// TwinCAT 3 PLC project plc_kfe_gatt
// ProgramVersion: 3.1.4023.0
// libraries:
//   LCLS General, * (SLAC)
//   lcls-twincat-motion, * (SLAC)
//   lcls-twincat-vacuum, * (SLAC)
//   PMPS, * (SLAC - LCLS)
//   Tc2_ControllerToolbox, * (Beckhoff Automation GmbH)
//   Tc2_EtherCAT, * (Beckhoff Automation GmbH)
//   Tc2_MC2, * (Beckhoff Automation GmbH)
//   Tc2_Standard, * (Beckhoff Automation GmbH)
//   Tc2_System, * (Beckhoff Automation GmbH)
//   Tc2_Utilities, * (Beckhoff Automation GmbH)
//   Tc3_JsonXml, * (Beckhoff Automation GmbH)
//   Tc3_Module, * (Beckhoff Automation GmbH)
//   TcUnit, * (www.tcunit.org)
// project tree:
//   DUTs/ E_HomeState.TcDUT (not stored), E_MAA_States.TcDUT (not stored), E_MoveState.TcDUT (not stored), ST_VGP.TcDUT (not stored)
//   GVLs/ GVL_Devices.TcGVL, GVL_GATT.TcGVL (not stored), GVL_ILK.TcGVL, GVL_MOT.TcGVL (not stored), GVL_Variables.TcGVL (not stored), Main.TcGVL (not stored)
//   / PlcTask.TcTTO (not stored)
//   POUs/ DIAGNOSTICS.TcPOU, FB_MAA.TcPOU, FB_MAA_States.TcPOU, FB_VGP.TcPOU, PRG_1_PlcTask.TcPOU, PRG_GATT.TcPOU, PRG_ILK.TcPOU, PRG_INJ.TcPOU, PRG_Motion.TcPOU, PRG_Motors_Test.TcPOU (not stored), PRG_VGP.TcPOU (not stored)
//   POUs/Test/ FB_ILK_TEST.TcPOU
// real-time tasks:
//   TASK PlcTask: cycle T#10ms, priority 20, ADS port 350
// motion (NC):
//   TASK NC-Task 1 SAF: cycle T#2ms, priority 4, ADS port 501
//   TASK NC-Task 1 SVB: cycle T#10ms, priority 8, ADS port 511
//   AXIS MA_1_X (id 1)
//     Velo: Maximum=5
//     OtherSettings: AllowMotionCmdToSlave=true
//     encoder EncType=4
//       EncPara: ScaleFactorNumerator=6.1991875e-05, MaxCount=#x0000ffff
//         Inc: RefSoftSyncMask=#x0000ffff
//     drive DrvType=24
//       Analog: VeloReferenz=7.93496, TorqueScale=10, ScaleFactorActTorque=0.1
//       TimeComp: TaskDelayCycles=1
//     controller CtrType=1
//       CtrPara: PriorControlFactor=1
//         Observer: BandWidth=20
//   AXIS MA_1_Y (id 2)
//     Dynamic: AccelerationMaximum=30, DecelerationMaximum=30
//     Velo: Maximum=40
//     OtherSettings: AllowMotionCmdToSlave=true
//     encoder EncType=7
//       EncPara: ScaleFactorNumerator=0.001452636719, Offset=-47.5985, MaxCount=#x0000ffff, ReferenceSystem=1
//         Inc: RefSoftSyncMask=#x0000ffff
//     drive DrvType=24
//       Analog: VeloReferenz=50, TorqueScale=10, ScaleFactorActTorque=0.1
//       TimeComp: TaskDelayCycles=1
//     controller CtrType=1
//       CtrPara: PriorControlFactor=1
//         Observer: BandWidth=20
//   AXIS MA_2_X (id 3)
//     Velo: Maximum=5
//     OtherSettings: AllowMotionCmdToSlave=true
//     encoder EncType=4
//       EncPara: ScaleFactorNumerator=6.1991875e-05, MaxCount=#x0000ffff
//         Inc: RefSoftSyncMask=#x0000ffff
//     drive DrvType=24
//       Analog: VeloReferenz=7.93496, TorqueScale=10, ScaleFactorActTorque=0.1
//       TimeComp: TaskDelayCycles=1
//     controller CtrType=1
//       CtrPara: PriorControlFactor=1
//         Observer: BandWidth=20
//   AXIS MA_2_Y (id 4)
//     Dynamic: AccelerationMaximum=30, DecelerationMaximum=30
//     Velo: Maximum=40
//     OtherSettings: AllowMotionCmdToSlave=true
//     encoder EncType=7
//       EncPara: ScaleFactorNumerator=0.001440429688, Offset=-47.056, MaxCount=#x0000ffff, ReferenceSystem=1
//         Inc: RefSoftSyncMask=#x0000ffff
//     drive DrvType=24
//       Analog: VeloReferenz=50, TorqueScale=10, ScaleFactorActTorque=0.1
//       TimeComp: TaskDelayCycles=1
//     controller CtrType=1
//       CtrPara: PriorControlFactor=1
//         Observer: BandWidth=20
//   AXIS MA_3_X (id 5)
//     Velo: Maximum=5
//     OtherSettings: AllowMotionCmdToSlave=true
//     encoder EncType=4
//       EncPara: ScaleFactorNumerator=6.1991875e-05, MaxCount=#x0000ffff
//         Inc: RefSoftSyncMask=#x0000ffff
//     drive DrvType=24
//       Analog: VeloReferenz=7.93496, TorqueScale=10, ScaleFactorActTorque=0.1
//       TimeComp: TaskDelayCycles=1
//     controller CtrType=1
//       CtrPara: PriorControlFactor=1
//         Observer: BandWidth=20
//   AXIS MA_3_Y (id 6)
//     Dynamic: AccelerationMaximum=30, DecelerationMaximum=30
//     Velo: Maximum=40
//     OtherSettings: AllowMotionCmdToSlave=true
//     encoder EncType=7
//       EncPara: ScaleFactorNumerator=0.001439703369, Offset=-47.15, MaxCount=#x0000ffff, ReferenceSystem=1
//         SoftEndMaxControl: Range=47.2
//         Inc: RefSoftSyncMask=#x0000ffff
//     drive DrvType=24
//       Analog: VeloReferenz=50, TorqueScale=10, ScaleFactorActTorque=0.1
//       TimeComp: TaskDelayCycles=1
//     controller CtrType=1
//       CtrPara: PriorControlFactor=1
//         PosDiffControl: Range=1.5
//         Observer: BandWidth=20
//   AXIS MA_4_X (id 7)
//     Velo: Maximum=5
//     OtherSettings: AllowMotionCmdToSlave=true
//     encoder EncType=4
//       EncPara: ScaleFactorNumerator=6.1991875e-05, MaxCount=#x0000ffff
//         Inc: RefSoftSyncMask=#x0000ffff
//     drive DrvType=24
//       Analog: VeloReferenz=7.93496, TorqueScale=10, ScaleFactorActTorque=0.1
//       TimeComp: TaskDelayCycles=1
//     controller CtrType=1
//       CtrPara: PriorControlFactor=1
//         Observer: BandWidth=20
//   AXIS MA_4_Y (id 8)
//     Dynamic: AccelerationMaximum=30, DecelerationMaximum=30
//     Velo: Maximum=40
//     OtherSettings: AllowMotionCmdToSlave=true
//     encoder EncType=4
//       EncPara: ScaleFactorNumerator=0.000390625, MaxCount=#x0000ffff
//         Inc: RefSoftSyncMask=#x0000ffff
//     drive DrvType=24
//       Analog: VeloReferenz=50, TorqueScale=10, ScaleFactorActTorque=0.1
//       TimeComp: TaskDelayCycles=1
//     controller CtrType=1
//       CtrPara: PriorControlFactor=1
//         Observer: BandWidth=20
//   AXIS VGP_80 (id 9)
//     Velo: Maximum=1800
//     OtherSettings: AllowMotionCmdToSlave=true
//     encoder EncType=4
//       EncPara: ScaleFactorNumerator=0.0390625, Inverse=true, MaxCount=#x0000ffff
//         SoftEndMinControl: Enable=true, Range=-15
//         SoftEndMaxControl: Enable=true, Range=1695
//         Inc: RefSoftSyncMask=#x0000ffff
//     drive DrvType=24
//       Analog: VeloReferenz=2000, TorqueScale=10, ScaleFactorActTorque=0.1
//       TimeComp: TaskDelayCycles=1
//     controller CtrType=1
//       CtrPara: PriorControlFactor=1
//         PosDiffControl: Range=75
//         Observer: BandWidth=20
// I/O:
//   DEVICE =+-CX2020%_2FEtherCAT1
// variable links:
//   NC-Task 1 SAF/Axes/MA_1_X <-> =+-CX2020/EtherCAT1/=+-EK1100_02_00/=+-ES7041_02_05
//     Drive/Inputs/In/nState1 @bit 3 <-> STM Status/Status/Error
//     Drive/Inputs/In/nState1 @bit 5 <-> STM Status/Status/Moving negative
//     Drive/Inputs/In/nState1 @bit 4 <-> STM Status/Status/Moving positive
//     Drive/Inputs/In/nState1 @bit 1 <-> STM Status/Status/Ready
//     Drive/Inputs/In/nState1 <-> STM Status/Status/Ready to enable
//     Drive/Inputs/In/nState1 @bit 6 <-> STM Status/Status/Torque reduced
//     Drive/Inputs/In/nState1 @bit 2 <-> STM Status/Status/Warning
//     Drive/Inputs/In/nState2 @bit 3 <-> STM Status/Status/Digital input 1
//     Drive/Inputs/In/nState2 @bit 4 <-> STM Status/Status/Digital input 2
//     Drive/Inputs/In/nState2 @bit 5 <-> STM Status/Status/Sync error
//     Drive/Inputs/In/nState2 @bit 7 <-> STM Status/Status/TxPDO Toggle
//     Drive/Inputs/In/nState4 @bit 1 <-> WcState/InputToggle
//     Drive/Inputs/In/nState4 <-> WcState/WcState
//     Drive/Outputs/Out/nCtrl1 <-> STM Control/Control/Enable
//     Drive/Outputs/Out/nCtrl1 @bit 2 <-> STM Control/Control/Reduce torque
//     Drive/Outputs/Out/nCtrl1 @bit 1 <-> STM Control/Control/Reset
//     Drive/Outputs/Out/nDataOut2[0] <-> STM Velocity/Velocity
//     Enc/Inputs/In/nDataIn1[0] <-> ENC Status compact/Counter value
//     Enc/Inputs/In/nDataIn2[0] <-> ENC Status compact/Latch value
//     Enc/Inputs/In/nState1 @bit 4 <-> ENC Status compact/Status/Counter overflow
//     Enc/Inputs/In/nState1 @bit 3 <-> ENC Status compact/Status/Counter underflow
//     Enc/Inputs/In/nState1 @bit 7 <-> ENC Status compact/Status/Extrapolation stall
//     Enc/Inputs/In/nState1 <-> ENC Status compact/Status/Latch C valid
//     Enc/Inputs/In/nState1 @bit 1 <-> ENC Status compact/Status/Latch extern valid
//     Enc/Inputs/In/nState1 @bit 2 <-> ENC Status compact/Status/Set counter done
//     Enc/Inputs/In/nState2 @bit 4 <-> ENC Status compact/Status/Status of extern latch
//     Enc/Inputs/In/nState2 <-> ENC Status compact/Status/Status of input A
//     Enc/Inputs/In/nState2 @bit 1 <-> ENC Status compact/Status/Status of input B
//     Enc/Inputs/In/nState2 @bit 2 <-> ENC Status compact/Status/Status of input C
//     Enc/Inputs/In/nState2 @bit 5 <-> ENC Status compact/Status/Sync error
//     Enc/Inputs/In/nState2 @bit 7 <-> ENC Status compact/Status/TxPDO Toggle
//     Enc/Inputs/In/nState4 @bit 1 <-> WcState/InputToggle
//     Enc/Inputs/In/nState4 <-> WcState/WcState
//     Enc/Outputs/Out/nCtrl1 <-> ENC Control compact/Control/Enable latch C
//     Enc/Outputs/Out/nCtrl1 @bit 3 <-> ENC Control compact/Control/Enable latch extern on negative edge
//     Enc/Outputs/Out/nCtrl1 @bit 1 <-> ENC Control compact/Control/Enable latch extern on positive edge
//     Enc/Outputs/Out/nCtrl1 @bit 2 <-> ENC Control compact/Control/Set counter
//     Enc/Outputs/Out/nDataOut1[0] <-> ENC Control compact/Set counter value
//   NC-Task 1 SAF/Axes/MA_1_Y <-> =+-CX2020/EtherCAT1/=+-EK1100_02_00/=+-ES3054_02_17
//     Enc/Inputs/In/nDataIn1[0] <-> AI Standard Channel 2/Value
//     Enc/Inputs/In/nState4 @bit 1 <-> WcState/InputToggle
//     Enc/Inputs/In/nState4 <-> WcState/WcState
//   NC-Task 1 SAF/Axes/MA_1_Y <-> =+-CX2020/EtherCAT1/=+-EK1100_02_00/=+-ES7041_02_06
//     Drive/Inputs/In/nState1 @bit 3 <-> STM Status/Status/Error
//     Drive/Inputs/In/nState1 @bit 5 <-> STM Status/Status/Moving negative
//     Drive/Inputs/In/nState1 @bit 4 <-> STM Status/Status/Moving positive
//     Drive/Inputs/In/nState1 @bit 1 <-> STM Status/Status/Ready
//     Drive/Inputs/In/nState1 <-> STM Status/Status/Ready to enable
//     Drive/Inputs/In/nState1 @bit 6 <-> STM Status/Status/Torque reduced
//     Drive/Inputs/In/nState1 @bit 2 <-> STM Status/Status/Warning
//     Drive/Inputs/In/nState2 @bit 3 <-> STM Status/Status/Digital input 1
//     Drive/Inputs/In/nState2 @bit 4 <-> STM Status/Status/Digital input 2
//     Drive/Inputs/In/nState2 @bit 5 <-> STM Status/Status/Sync error
//     Drive/Inputs/In/nState2 @bit 7 <-> STM Status/Status/TxPDO Toggle
//     Drive/Inputs/In/nState4 @bit 1 <-> WcState/InputToggle
//     Drive/Inputs/In/nState4 <-> WcState/WcState
//     Drive/Outputs/Out/nCtrl1 <-> STM Control/Control/Enable
//     Drive/Outputs/Out/nCtrl1 @bit 2 <-> STM Control/Control/Reduce torque
//     Drive/Outputs/Out/nCtrl1 @bit 1 <-> STM Control/Control/Reset
//     Drive/Outputs/Out/nDataOut2[0] <-> STM Velocity/Velocity
//   NC-Task 1 SAF/Axes/MA_2_X <-> =+-CX2020/EtherCAT1/=+-EK1100_02_00/=+-ES7041_02_09
//     Drive/Inputs/In/nState1 @bit 3 <-> STM Status/Status/Error
//     Drive/Inputs/In/nState1 @bit 5 <-> STM Status/Status/Moving negative
//     Drive/Inputs/In/nState1 @bit 4 <-> STM Status/Status/Moving positive
//     Drive/Inputs/In/nState1 @bit 1 <-> STM Status/Status/Ready
//     Drive/Inputs/In/nState1 <-> STM Status/Status/Ready to enable
//     Drive/Inputs/In/nState1 @bit 6 <-> STM Status/Status/Torque reduced
//     Drive/Inputs/In/nState1 @bit 2 <-> STM Status/Status/Warning
//     Drive/Inputs/In/nState2 @bit 3 <-> STM Status/Status/Digital input 1
//     Drive/Inputs/In/nState2 @bit 4 <-> STM Status/Status/Digital input 2
//     Drive/Inputs/In/nState2 @bit 5 <-> STM Status/Status/Sync error
//     Drive/Inputs/In/nState2 @bit 7 <-> STM Status/Status/TxPDO Toggle
//     Drive/Inputs/In/nState4 @bit 1 <-> WcState/InputToggle
//     Drive/Inputs/In/nState4 <-> WcState/WcState
//     Drive/Outputs/Out/nCtrl1 <-> STM Control/Control/Enable
//     Drive/Outputs/Out/nCtrl1 @bit 2 <-> STM Control/Control/Reduce torque
//     Drive/Outputs/Out/nCtrl1 @bit 1 <-> STM Control/Control/Reset
//     Drive/Outputs/Out/nDataOut2[0] <-> STM Velocity/Velocity
//     Enc/Inputs/In/nDataIn1[0] <-> ENC Status compact/Counter value
//     Enc/Inputs/In/nDataIn2[0] <-> ENC Status compact/Latch value
//     Enc/Inputs/In/nState1 @bit 4 <-> ENC Status compact/Status/Counter overflow
//     Enc/Inputs/In/nState1 @bit 3 <-> ENC Status compact/Status/Counter underflow
//     Enc/Inputs/In/nState1 @bit 7 <-> ENC Status compact/Status/Extrapolation stall
//     Enc/Inputs/In/nState1 <-> ENC Status compact/Status/Latch C valid
//     Enc/Inputs/In/nState1 @bit 1 <-> ENC Status compact/Status/Latch extern valid
//     Enc/Inputs/In/nState1 @bit 2 <-> ENC Status compact/Status/Set counter done
//     Enc/Inputs/In/nState2 @bit 4 <-> ENC Status compact/Status/Status of extern latch
//     Enc/Inputs/In/nState2 <-> ENC Status compact/Status/Status of input A
//     Enc/Inputs/In/nState2 @bit 1 <-> ENC Status compact/Status/Status of input B
//     Enc/Inputs/In/nState2 @bit 2 <-> ENC Status compact/Status/Status of input C
//     Enc/Inputs/In/nState2 @bit 5 <-> ENC Status compact/Status/Sync error
//     Enc/Inputs/In/nState2 @bit 7 <-> ENC Status compact/Status/TxPDO Toggle
//     Enc/Inputs/In/nState4 @bit 1 <-> WcState/InputToggle
//     Enc/Inputs/In/nState4 <-> WcState/WcState
//     Enc/Outputs/Out/nCtrl1 <-> ENC Control compact/Control/Enable latch C
//     Enc/Outputs/Out/nCtrl1 @bit 3 <-> ENC Control compact/Control/Enable latch extern on negative edge
//     Enc/Outputs/Out/nCtrl1 @bit 1 <-> ENC Control compact/Control/Enable latch extern on positive edge
//     Enc/Outputs/Out/nCtrl1 @bit 2 <-> ENC Control compact/Control/Set counter
//     Enc/Outputs/Out/nDataOut1[0] <-> ENC Control compact/Set counter value
//   NC-Task 1 SAF/Axes/MA_2_Y <-> =+-CX2020/EtherCAT1/=+-EK1100_02_00/=+-ES3054_02_17
//     Enc/Inputs/In/nDataIn1[0] <-> AI Standard Channel 4/Value
//     Enc/Inputs/In/nState4 @bit 1 <-> WcState/InputToggle
//     Enc/Inputs/In/nState4 <-> WcState/WcState
//   NC-Task 1 SAF/Axes/MA_2_Y <-> =+-CX2020/EtherCAT1/=+-EK1100_02_00/=+-ES7041_02_10
//     Drive/Inputs/In/nState1 @bit 3 <-> STM Status/Status/Error
//     Drive/Inputs/In/nState1 @bit 5 <-> STM Status/Status/Moving negative
//     Drive/Inputs/In/nState1 @bit 4 <-> STM Status/Status/Moving positive
//     Drive/Inputs/In/nState1 @bit 1 <-> STM Status/Status/Ready
//     Drive/Inputs/In/nState1 <-> STM Status/Status/Ready to enable
//     Drive/Inputs/In/nState1 @bit 6 <-> STM Status/Status/Torque reduced
//     Drive/Inputs/In/nState1 @bit 2 <-> STM Status/Status/Warning
//     Drive/Inputs/In/nState2 @bit 3 <-> STM Status/Status/Digital input 1
//     Drive/Inputs/In/nState2 @bit 4 <-> STM Status/Status/Digital input 2
//     Drive/Inputs/In/nState2 @bit 5 <-> STM Status/Status/Sync error
//     Drive/Inputs/In/nState2 @bit 7 <-> STM Status/Status/TxPDO Toggle
//     Drive/Inputs/In/nState4 @bit 1 <-> WcState/InputToggle
//     Drive/Inputs/In/nState4 <-> WcState/WcState
//     Drive/Outputs/Out/nCtrl1 <-> STM Control/Control/Enable
//     Drive/Outputs/Out/nCtrl1 @bit 2 <-> STM Control/Control/Reduce torque
//     Drive/Outputs/Out/nCtrl1 @bit 1 <-> STM Control/Control/Reset
//     Drive/Outputs/Out/nDataOut2[0] <-> STM Velocity/Velocity
//   NC-Task 1 SAF/Axes/MA_3_X <-> =+-CX2020/EtherCAT1/=+-EK1100_04_00/=+-EL7041_04_07
//     Drive/Inputs/In/nState1 @bit 3 <-> STM Status/Status/Error
//     Drive/Inputs/In/nState1 @bit 5 <-> STM Status/Status/Moving negative
//     Drive/Inputs/In/nState1 @bit 4 <-> STM Status/Status/Moving positive
//     Drive/Inputs/In/nState1 @bit 1 <-> STM Status/Status/Ready
//     Drive/Inputs/In/nState1 <-> STM Status/Status/Ready to enable
//     Drive/Inputs/In/nState1 @bit 6 <-> STM Status/Status/Torque reduced
//     Drive/Inputs/In/nState1 @bit 2 <-> STM Status/Status/Warning
//     Drive/Inputs/In/nState2 @bit 3 <-> STM Status/Status/Digital input 1
//     Drive/Inputs/In/nState2 @bit 4 <-> STM Status/Status/Digital input 2
//     Drive/Inputs/In/nState2 @bit 5 <-> STM Status/Status/Sync error
//     Drive/Inputs/In/nState2 @bit 7 <-> STM Status/Status/TxPDO Toggle
//     Drive/Inputs/In/nState4 @bit 1 <-> WcState/InputToggle
//     Drive/Inputs/In/nState4 <-> WcState/WcState
//     Drive/Outputs/Out/nCtrl1 <-> STM Control/Control/Enable
//     Drive/Outputs/Out/nCtrl1 @bit 2 <-> STM Control/Control/Reduce torque
//     Drive/Outputs/Out/nCtrl1 @bit 1 <-> STM Control/Control/Reset
//     Drive/Outputs/Out/nDataOut2[0] <-> STM Velocity/Velocity
//     Enc/Inputs/In/nDataIn1[0] <-> ENC Status compact/Counter value
//     Enc/Inputs/In/nDataIn2[0] <-> ENC Status compact/Latch value
//     Enc/Inputs/In/nState1 @bit 4 <-> ENC Status compact/Status/Counter overflow
//     Enc/Inputs/In/nState1 @bit 3 <-> ENC Status compact/Status/Counter underflow
//     Enc/Inputs/In/nState1 @bit 7 <-> ENC Status compact/Status/Extrapolation stall
//     Enc/Inputs/In/nState1 <-> ENC Status compact/Status/Latch C valid
//     Enc/Inputs/In/nState1 @bit 1 <-> ENC Status compact/Status/Latch extern valid
//     Enc/Inputs/In/nState1 @bit 2 <-> ENC Status compact/Status/Set counter done
//     Enc/Inputs/In/nState2 @bit 4 <-> ENC Status compact/Status/Status of extern latch
//     Enc/Inputs/In/nState2 <-> ENC Status compact/Status/Status of input A
//     Enc/Inputs/In/nState2 @bit 1 <-> ENC Status compact/Status/Status of input B
//     Enc/Inputs/In/nState2 @bit 2 <-> ENC Status compact/Status/Status of input C
//     Enc/Inputs/In/nState2 @bit 5 <-> ENC Status compact/Status/Sync error
//     Enc/Inputs/In/nState2 @bit 7 <-> ENC Status compact/Status/TxPDO Toggle
//     Enc/Inputs/In/nState4 @bit 1 <-> WcState/InputToggle
//     Enc/Inputs/In/nState4 <-> WcState/WcState
//     Enc/Outputs/Out/nCtrl1 <-> ENC Control compact/Control/Enable latch C
//     Enc/Outputs/Out/nCtrl1 @bit 3 <-> ENC Control compact/Control/Enable latch extern on negative edge
//     Enc/Outputs/Out/nCtrl1 @bit 1 <-> ENC Control compact/Control/Enable latch extern on positive edge
//     Enc/Outputs/Out/nCtrl1 @bit 2 <-> ENC Control compact/Control/Set counter
//     Enc/Outputs/Out/nDataOut1[0] <-> ENC Control compact/Set counter value
//   NC-Task 1 SAF/Axes/MA_3_Y <-> =+-CX2020/EtherCAT1/=+-EK1100_04_00/=+-EL7041_04_08
//     Drive/Inputs/In/nState1 @bit 3 <-> STM Status/Status/Error
//     Drive/Inputs/In/nState1 @bit 5 <-> STM Status/Status/Moving negative
//     Drive/Inputs/In/nState1 @bit 4 <-> STM Status/Status/Moving positive
//     Drive/Inputs/In/nState1 @bit 1 <-> STM Status/Status/Ready
//     Drive/Inputs/In/nState1 <-> STM Status/Status/Ready to enable
//     Drive/Inputs/In/nState1 @bit 6 <-> STM Status/Status/Torque reduced
//     Drive/Inputs/In/nState1 @bit 2 <-> STM Status/Status/Warning
//     Drive/Inputs/In/nState2 @bit 3 <-> STM Status/Status/Digital input 1
//     Drive/Inputs/In/nState2 @bit 4 <-> STM Status/Status/Digital input 2
//     Drive/Inputs/In/nState2 @bit 5 <-> STM Status/Status/Sync error
//     Drive/Inputs/In/nState2 @bit 7 <-> STM Status/Status/TxPDO Toggle
//     Drive/Inputs/In/nState4 @bit 1 <-> WcState/InputToggle
//     Drive/Inputs/In/nState4 <-> WcState/WcState
//     Drive/Outputs/Out/nCtrl1 <-> STM Control/Control/Enable
//     Drive/Outputs/Out/nCtrl1 @bit 2 <-> STM Control/Control/Reduce torque
//     Drive/Outputs/Out/nCtrl1 @bit 1 <-> STM Control/Control/Reset
//     Drive/Outputs/Out/nDataOut2[0] <-> STM Velocity/Velocity
//   NC-Task 1 SAF/Axes/MA_3_Y <-> =+-CX2020/EtherCAT1/=+-EK1100_04_00/=+-ES3054_04_12
//     Enc/Inputs/In/nDataIn1[0] <-> AI Standard Channel 2/Value
//     Enc/Inputs/In/nState4 @bit 1 <-> WcState/InputToggle
//     Enc/Inputs/In/nState4 <-> WcState/WcState
//   NC-Task 1 SAF/Axes/MA_4_X <-> =+-CX2020/EtherCAT1/=+-EK1100_04_00/=+-EL7041_04_10
//     Drive/Inputs/In/nState1 @bit 3 <-> STM Status/Status/Error
//     Drive/Inputs/In/nState1 @bit 5 <-> STM Status/Status/Moving negative
//     Drive/Inputs/In/nState1 @bit 4 <-> STM Status/Status/Moving positive
//     Drive/Inputs/In/nState1 @bit 1 <-> STM Status/Status/Ready
//     Drive/Inputs/In/nState1 <-> STM Status/Status/Ready to enable
//     Drive/Inputs/In/nState1 @bit 6 <-> STM Status/Status/Torque reduced
//     Drive/Inputs/In/nState1 @bit 2 <-> STM Status/Status/Warning
//     Drive/Inputs/In/nState2 @bit 3 <-> STM Status/Status/Digital input 1
//     Drive/Inputs/In/nState2 @bit 4 <-> STM Status/Status/Digital input 2
//     Drive/Inputs/In/nState2 @bit 5 <-> STM Status/Status/Sync error
//     Drive/Inputs/In/nState2 @bit 7 <-> STM Status/Status/TxPDO Toggle
//     Drive/Inputs/In/nState4 @bit 1 <-> WcState/InputToggle
//     Drive/Inputs/In/nState4 <-> WcState/WcState
//     Drive/Outputs/Out/nCtrl1 <-> STM Control/Control/Enable
//     Drive/Outputs/Out/nCtrl1 @bit 2 <-> STM Control/Control/Reduce torque
//     Drive/Outputs/Out/nCtrl1 @bit 1 <-> STM Control/Control/Reset
//     Drive/Outputs/Out/nDataOut2[0] <-> STM Velocity/Velocity
//     Enc/Inputs/In/nDataIn1[0] <-> ENC Status compact/Counter value
//     Enc/Inputs/In/nDataIn2[0] <-> ENC Status compact/Latch value
//     Enc/Inputs/In/nState1 @bit 4 <-> ENC Status compact/Status/Counter overflow
//     Enc/Inputs/In/nState1 @bit 3 <-> ENC Status compact/Status/Counter underflow
//     Enc/Inputs/In/nState1 @bit 7 <-> ENC Status compact/Status/Extrapolation stall
//     Enc/Inputs/In/nState1 <-> ENC Status compact/Status/Latch C valid
//     Enc/Inputs/In/nState1 @bit 1 <-> ENC Status compact/Status/Latch extern valid
//     Enc/Inputs/In/nState1 @bit 2 <-> ENC Status compact/Status/Set counter done
//     Enc/Inputs/In/nState2 @bit 4 <-> ENC Status compact/Status/Status of extern latch
//     Enc/Inputs/In/nState2 <-> ENC Status compact/Status/Status of input A
//     Enc/Inputs/In/nState2 @bit 1 <-> ENC Status compact/Status/Status of input B
//     Enc/Inputs/In/nState2 @bit 2 <-> ENC Status compact/Status/Status of input C
//     Enc/Inputs/In/nState2 @bit 5 <-> ENC Status compact/Status/Sync error
//     Enc/Inputs/In/nState2 @bit 7 <-> ENC Status compact/Status/TxPDO Toggle
//     Enc/Inputs/In/nState4 @bit 1 <-> WcState/InputToggle
//     Enc/Inputs/In/nState4 <-> WcState/WcState
//     Enc/Outputs/Out/nCtrl1 <-> ENC Control compact/Control/Enable latch C
//     Enc/Outputs/Out/nCtrl1 @bit 3 <-> ENC Control compact/Control/Enable latch extern on negative edge
//     Enc/Outputs/Out/nCtrl1 @bit 1 <-> ENC Control compact/Control/Enable latch extern on positive edge
//     Enc/Outputs/Out/nCtrl1 @bit 2 <-> ENC Control compact/Control/Set counter
//     Enc/Outputs/Out/nDataOut1[0] <-> ENC Control compact/Set counter value
//   NC-Task 1 SAF/Axes/MA_4_Y <-> =+-CX2020/EtherCAT1/=+-EK1100_04_00/=+-EL7041_04_11
//     Drive/Inputs/In/nState1 @bit 3 <-> STM Status/Status/Error
//     Drive/Inputs/In/nState1 @bit 5 <-> STM Status/Status/Moving negative
//     Drive/Inputs/In/nState1 @bit 4 <-> STM Status/Status/Moving positive
//     Drive/Inputs/In/nState1 @bit 1 <-> STM Status/Status/Ready
//     Drive/Inputs/In/nState1 <-> STM Status/Status/Ready to enable
//     Drive/Inputs/In/nState1 @bit 6 <-> STM Status/Status/Torque reduced
//     Drive/Inputs/In/nState1 @bit 2 <-> STM Status/Status/Warning
//     Drive/Inputs/In/nState2 @bit 3 <-> STM Status/Status/Digital input 1
//     Drive/Inputs/In/nState2 @bit 4 <-> STM Status/Status/Digital input 2
//     Drive/Inputs/In/nState2 @bit 5 <-> STM Status/Status/Sync error
//     Drive/Inputs/In/nState2 @bit 7 <-> STM Status/Status/TxPDO Toggle
//     Drive/Inputs/In/nState4 @bit 1 <-> WcState/InputToggle
//     Drive/Inputs/In/nState4 <-> WcState/WcState
//     Drive/Outputs/Out/nCtrl1 <-> STM Control/Control/Enable
//     Drive/Outputs/Out/nCtrl1 @bit 2 <-> STM Control/Control/Reduce torque
//     Drive/Outputs/Out/nCtrl1 @bit 1 <-> STM Control/Control/Reset
//     Drive/Outputs/Out/nDataOut2[0] <-> STM Velocity/Velocity
//     Enc/Inputs/In/nDataIn1[0] <-> ENC Status compact/Counter value
//     Enc/Inputs/In/nDataIn2[0] <-> ENC Status compact/Latch value
//     Enc/Inputs/In/nState1 @bit 4 <-> ENC Status compact/Status/Counter overflow
//     Enc/Inputs/In/nState1 @bit 3 <-> ENC Status compact/Status/Counter underflow
//     Enc/Inputs/In/nState1 @bit 7 <-> ENC Status compact/Status/Extrapolation stall
//     Enc/Inputs/In/nState1 <-> ENC Status compact/Status/Latch C valid
//     Enc/Inputs/In/nState1 @bit 1 <-> ENC Status compact/Status/Latch extern valid
//     Enc/Inputs/In/nState1 @bit 2 <-> ENC Status compact/Status/Set counter done
//     Enc/Inputs/In/nState2 @bit 4 <-> ENC Status compact/Status/Status of extern latch
//     Enc/Inputs/In/nState2 <-> ENC Status compact/Status/Status of input A
//     Enc/Inputs/In/nState2 @bit 1 <-> ENC Status compact/Status/Status of input B
//     Enc/Inputs/In/nState2 @bit 2 <-> ENC Status compact/Status/Status of input C
//     Enc/Inputs/In/nState2 @bit 5 <-> ENC Status compact/Status/Sync error
//     Enc/Inputs/In/nState2 @bit 7 <-> ENC Status compact/Status/TxPDO Toggle
//     Enc/Inputs/In/nState4 @bit 1 <-> WcState/InputToggle
//     Enc/Inputs/In/nState4 <-> WcState/WcState
//     Enc/Outputs/Out/nCtrl1 <-> ENC Control compact/Control/Enable latch C
//     Enc/Outputs/Out/nCtrl1 @bit 3 <-> ENC Control compact/Control/Enable latch extern on negative edge
//     Enc/Outputs/Out/nCtrl1 @bit 1 <-> ENC Control compact/Control/Enable latch extern on positive edge
//     Enc/Outputs/Out/nCtrl1 @bit 2 <-> ENC Control compact/Control/Set counter
//     Enc/Outputs/Out/nDataOut1[0] <-> ENC Control compact/Set counter value
//   NC-Task 1 SAF/Axes/VGP_80 <-> =+-CX2020/EtherCAT1/=+-EK1100_04_00/=+-EL5101_04_05
//     Enc/Inputs/In/nDataIn1[0] <-> ENC Status compact/Counter value
//     Enc/Inputs/In/nDataIn2[0] <-> ENC Status compact/Latch value
//     Enc/Inputs/In/nState1 @bit 4 <-> ENC Status compact/Status/Counter overflow
//     Enc/Inputs/In/nState1 @bit 3 <-> ENC Status compact/Status/Counter underflow
//     Enc/Inputs/In/nState1 @bit 7 <-> ENC Status compact/Status/Extrapolation stall
//     Enc/Inputs/In/nState1 <-> ENC Status compact/Status/Latch C valid
//     Enc/Inputs/In/nState1 @bit 1 <-> ENC Status compact/Status/Latch extern valid
//     Enc/Inputs/In/nState1 @bit 6 <-> ENC Status compact/Status/Open circuit
//     Enc/Inputs/In/nState1 @bit 2 <-> ENC Status compact/Status/Set counter done
//     Enc/Inputs/In/nState1 @bit 5 <-> ENC Status compact/Status/Status of input status
//     Enc/Inputs/In/nState2 @bit 4 <-> ENC Status compact/Status/Status of extern latch
//     Enc/Inputs/In/nState2 <-> ENC Status compact/Status/Status of input A
//     Enc/Inputs/In/nState2 @bit 1 <-> ENC Status compact/Status/Status of input B
//     Enc/Inputs/In/nState2 @bit 2 <-> ENC Status compact/Status/Status of input C
//     Enc/Inputs/In/nState2 @bit 3 <-> ENC Status compact/Status/Status of input gate
//     Enc/Inputs/In/nState2 @bit 5 <-> ENC Status compact/Status/Sync error
//     Enc/Inputs/In/nState2 @bit 6 <-> ENC Status compact/Status/TxPDO State
//     Enc/Inputs/In/nState2 @bit 7 <-> ENC Status compact/Status/TxPDO Toggle
//     Enc/Inputs/In/nState4 @bit 1 <-> WcState/InputToggle
//     Enc/Inputs/In/nState4 <-> WcState/WcState
//     Enc/Outputs/Out/nCtrl1 <-> ENC Control compact/Control/Enable latch C
//     Enc/Outputs/Out/nCtrl1 @bit 3 <-> ENC Control compact/Control/Enable latch extern on negative edge
//     Enc/Outputs/Out/nCtrl1 @bit 1 <-> ENC Control compact/Control/Enable latch extern on positive edge
//     Enc/Outputs/Out/nCtrl1 @bit 2 <-> ENC Control compact/Control/Set counter
//     Enc/Outputs/Out/nDataOut1[0] <-> ENC Control compact/Set counter value
//   NC-Task 1 SAF/Axes/VGP_80 <-> =+-CX2020/EtherCAT1/=+-EK1100_04_00/=+-EL7041_04_04
//     Drive/Inputs/In/nState1 @bit 3 <-> STM Status/Status/Error
//     Drive/Inputs/In/nState1 @bit 5 <-> STM Status/Status/Moving negative
//     Drive/Inputs/In/nState1 @bit 4 <-> STM Status/Status/Moving positive
//     Drive/Inputs/In/nState1 @bit 1 <-> STM Status/Status/Ready
//     Drive/Inputs/In/nState1 <-> STM Status/Status/Ready to enable
//     Drive/Inputs/In/nState1 @bit 6 <-> STM Status/Status/Torque reduced
//     Drive/Inputs/In/nState1 @bit 2 <-> STM Status/Status/Warning
//     Drive/Inputs/In/nState2 @bit 3 <-> STM Status/Status/Digital input 1
//     Drive/Inputs/In/nState2 @bit 4 <-> STM Status/Status/Digital input 2
//     Drive/Inputs/In/nState2 @bit 5 <-> STM Status/Status/Sync error
//     Drive/Inputs/In/nState2 @bit 7 <-> STM Status/Status/TxPDO Toggle
//     Drive/Inputs/In/nState4 @bit 1 <-> WcState/InputToggle
//     Drive/Inputs/In/nState4 <-> WcState/WcState
//     Drive/Outputs/Out/nCtrl1 <-> STM Control/Control/Enable
//     Drive/Outputs/Out/nCtrl1 @bit 2 <-> STM Control/Control/Reduce torque
//     Drive/Outputs/Out/nCtrl1 @bit 1 <-> STM Control/Control/Reset
//     Drive/Outputs/Out/nDataOut2[0] <-> STM Velocity/Velocity
//   plc_kfe_gatt Instance <-> =+-CX2020/EtherCAT1/=+-EK1100_01_00/=+-EL2798_01_03
//     PlcTask Outputs/GVL_Devices.fb_AT1K0_GAS_GCC_10.q_xHV_DIS <-> Channel 1/fb_AT1K0_GAS_GCC_10.q_xHV_DIS
//     PlcTask Outputs/GVL_Devices.fb_AT1K0_GAS_GCC_20.q_xHV_DIS <-> Channel 2/fb_AT1K0_GAS_GCC_20.q_xHV_DIS
//     PlcTask Outputs/GVL_Devices.fb_AT1K0_GAS_GCC_30.q_xHV_DIS <-> Channel 5/fb_AT1K0_GAS_GCC_30.q_xHV_DIS
//     PlcTask Outputs/GVL_Devices.fb_AT1K0_GAS_GCC_40.q_xHV_DIS <-> Channel 6/fb_AT1K0_GAS_GCC_40.q_xHV_DIS
//   plc_kfe_gatt Instance <-> =+-CX2020/EtherCAT1/=+-EK1100_01_00/=+-EL2798_01_08
//     PlcTask Outputs/GVL_Devices.fb_AT1K0_GAS_GCC_50.q_xHV_DIS <-> Channel 1/fb_AT1K0_GAS_GCC_50.q_xHV_DIS
//     PlcTask Outputs/GVL_Devices.fb_AT1K0_GAS_GCC_60.q_xHV_DIS <-> Channel 2/fb_AT1K0_GAS_GCC_60.q_xHV_DIS
//     PlcTask Outputs/GVL_Devices.fb_AT1K0_GAS_GCC_80.q_xHV_DIS <-> Channel 5/fb_AT1K0_GAS_GCC_80.q_xHV_DIS
//   plc_kfe_gatt Instance <-> =+-CX2020/EtherCAT1/=+-EK1100_01_00/=+-EL2798_01_14
//     PlcTask Outputs/GVL_Devices.fb_AT1K0_GAS_GCC_100.q_xHV_DIS <-> Channel 2/fb_AT1K0_GAS_GCC_100.q_xHV_DIS
//     PlcTask Outputs/GVL_Devices.fb_AT1K0_GAS_GCC_110.q_xHV_DIS <-> Channel 5/fb_AT1K0_GAS_GCC_110.q_xHV_DIS
//     PlcTask Outputs/GVL_Devices.fb_AT1K0_GAS_GCC_120.q_xHV_DIS <-> Channel 6/fb_AT1K0_GAS_GCC_120.q_xHV_DIS
//     PlcTask Outputs/GVL_Devices.fb_AT1K0_GAS_GCC_90.q_xHV_DIS <-> Channel 1/fb_AT1K0_GAS_GCC_90.q_xHV_DIS
//   plc_kfe_gatt Instance <-> =+-CX2020/EtherCAT1/=+-EK1100_01_00/=+-EL2798_01_19
//     PlcTask Outputs/GVL_Devices.fb_AT1K0_GAS_GCC_130.q_xHV_DIS <-> Channel 1/Output
//     PlcTask Outputs/GVL_Devices.fb_AT1K0_GAS_GCC_140.q_xHV_DIS <-> Channel 2/Output
//   plc_kfe_gatt Instance <-> =+-CX2020/EtherCAT1/=+-EK1100_01_00/=+-ES3064_01_01
//     PlcTask Inputs/GVL_Devices.fb_AT1K0_GAS_GCC_10.i_iPRESS_R <-> AI Standard Channel 1/fb_AT1K0_GAS_GCC_10.i_iPRESS_R
//     PlcTask Inputs/GVL_Devices.fb_AT1K0_GAS_GCC_20.i_iPRESS_R <-> AI Standard Channel 3/fb_AT1K0_GAS_GCC_20.i_iPRESS_R
//   plc_kfe_gatt Instance <-> =+-CX2020/EtherCAT1/=+-EK1100_01_00/=+-ES3064_01_02
//     PlcTask Inputs/GVL_Devices.fb_AT1K0_GAS_GPI_10.i_iPRESS_R <-> AI Standard Channel 1/fb_AT1K0_GAS_GPI_10.i_iPRESS_R
//     PlcTask Inputs/GVL_Devices.fb_AT1K0_GAS_GPI_20.i_iPRESS_R <-> AI Standard Channel 2/fb_AT1K0_GAS_GPI_20.i_iPRESS_R
//   plc_kfe_gatt Instance <-> =+-CX2020/EtherCAT1/=+-EK1100_01_00/=+-ES3064_01_04
//     PlcTask Inputs/GVL_Devices.fb_AT1K0_GAS_GCC_30.i_iPRESS_R <-> AI Standard Channel 1/fb_AT1K0_GAS_GCC_30.i_iPRESS_R
//     PlcTask Inputs/GVL_Devices.fb_AT1K0_GAS_GCC_40.i_iPRESS_R <-> AI Standard Channel 3/fb_AT1K0_GAS_GCC_40.i_iPRESS_R
//   plc_kfe_gatt Instance <-> =+-CX2020/EtherCAT1/=+-EK1100_01_00/=+-ES3064_01_05
//     PlcTask Inputs/GVL_Devices.fb_AT1K0_GAS_GPI_30.i_iPRESS_R <-> AI Standard Channel 1/fb_AT1K0_GAS_GPI_30.i_iPRESS_R
//     PlcTask Inputs/GVL_Devices.fb_AT1K0_GAS_GPI_40.i_iPRESS_R <-> AI Standard Channel 2/fb_AT1K0_GAS_GPI_40.i_iPRESS_R
//   plc_kfe_gatt Instance <-> =+-CX2020/EtherCAT1/=+-EK1100_01_00/=+-ES3064_01_06
//     PlcTask Inputs/GVL_Devices.fb_AT1K0_GAS_GCC_50.i_iPRESS_R <-> AI Standard Channel 1/fb_AT1K0_GAS_GCC_50.i_iPRESS_R
//     PlcTask Inputs/GVL_Devices.fb_AT1K0_GAS_GCC_60.i_iPRESS_R <-> AI Standard Channel 3/fb_AT1K0_GAS_GCC_60.i_iPRESS_R
//   plc_kfe_gatt Instance <-> =+-CX2020/EtherCAT1/=+-EK1100_01_00/=+-ES3064_01_07
//     PlcTask Inputs/GVL_Devices.fb_AT1K0_GAS_GPI_50.i_iPRESS_R <-> AI Standard Channel 1/fb_AT1K0_GAS_GPI_50.i_iPRESS_R
//     PlcTask Inputs/GVL_Devices.fb_AT1K0_GAS_GPI_60.i_iPRESS_R <-> AI Standard Channel 2/fb_AT1K0_GAS_GPI_60.i_iPRESS_R
//   plc_kfe_gatt Instance <-> =+-CX2020/EtherCAT1/=+-EK1100_01_00/=+-ES3064_01_09
//     PlcTask Inputs/GVL_Devices.fb_AT1K0_GAS_GCC_80.i_iPRESS_R <-> AI Standard Channel 1/fb_AT1K0_GAS_GCC_80.i_iPRESS_R
//     PlcTask Inputs/GVL_Devices.fb_AT1K0_GAS_GPI_80.i_iPRESS_R <-> AI Standard Channel 3/fb_AT1K0_GAS_GPI_80.i_iPRESS_R
//   plc_kfe_gatt Instance <-> =+-CX2020/EtherCAT1/=+-EK1100_01_00/=+-ES3064_01_10
//     PlcTask Inputs/GVL_Devices.fb_AT1K0_GAS_GPI_11.i_iPRESS_R <-> AI Standard Channel 1/fb_AT1K0_GAS_GPI_11.i_iPRESS_R
//     PlcTask Inputs/GVL_Devices.fb_AT1K0_GAS_GPI_51.i_iPRESS_R <-> AI Standard Channel 2/fb_AT1K0_GAS_GPI_51.i_iPRESS_R
//   plc_kfe_gatt Instance <-> =+-CX2020/EtherCAT1/=+-EK1100_01_00/=+-ES3064_01_12
//     PlcTask Inputs/GVL_Devices.fb_AT1K0_GAS_GCC_100.i_iPRESS_R <-> AI Standard Channel 3/fb_AT1K0_GAS_GCC_100.i_iPRESS_R
//     PlcTask Inputs/GVL_Devices.fb_AT1K0_GAS_GCC_90.i_iPRESS_R <-> AI Standard Channel 1/fb_AT1K0_GAS_GCC_90.i_iPRESS_R
//   plc_kfe_gatt Instance <-> =+-CX2020/EtherCAT1/=+-EK1100_01_00/=+-ES3064_01_13
//     PlcTask Inputs/GVL_Devices.fb_AT1K0_GAS_GPI_100.i_iPRESS_R <-> AI Standard Channel 2/fb_AT1K0_GAS_GPI_100.i_iPRESS_R
//     PlcTask Inputs/GVL_Devices.fb_AT1K0_GAS_GPI_90.i_iPRESS_R <-> AI Standard Channel 1/fb_AT1K0_GAS_GPI_90.i_iPRESS_R
//   plc_kfe_gatt Instance <-> =+-CX2020/EtherCAT1/=+-EK1100_01_00/=+-ES3064_01_15
//     PlcTask Inputs/GVL_Devices.fb_AT1K0_GAS_GCC_110.i_iPRESS_R <-> AI Standard Channel 1/fb_AT1K0_GAS_GCC_110.i_iPRESS_R
//     PlcTask Inputs/GVL_Devices.fb_AT1K0_GAS_GCC_120.i_iPRESS_R <-> AI Standard Channel 3/fb_AT1K0_GAS_GCC_120.i_iPRESS_R
//   plc_kfe_gatt Instance <-> =+-CX2020/EtherCAT1/=+-EK1100_01_00/=+-ES3064_01_16
//     PlcTask Inputs/GVL_Devices.fb_AT1K0_GAS_GPI_110.i_iPRESS_R <-> AI Standard Channel 1/fb_AT1K0_GAS_GPI_110.i_iPRESS_R
//     PlcTask Inputs/GVL_Devices.fb_AT1K0_GAS_GPI_120.i_iPRESS_R <-> AI Standard Channel 2/fb_AT1K0_GAS_GPI_120.i_iPRESS_R
//   plc_kfe_gatt Instance <-> =+-CX2020/EtherCAT1/=+-EK1100_01_00/=+-ES3064_01_17
//     PlcTask Inputs/GVL_Devices.fb_AT1K0_GAS_GCC_130.i_iPRESS_R <-> AI Standard Channel 1/fb_AT1K0_GAS_GCC_130.i_iPRESS_R
//     PlcTask Inputs/GVL_Devices.fb_AT1K0_GAS_GCC_140.i_iPRESS_R <-> AI Standard Channel 3/fb_AT1K0_GAS_GCC_140.i_iPRESS_R
//   plc_kfe_gatt Instance <-> =+-CX2020/EtherCAT1/=+-EK1100_01_00/=+-ES3064_01_18
//     PlcTask Inputs/GVL_Devices.fb_AT1K0_GAS_GPI_130.i_iPRESS_R <-> AI Standard Channel 1/fb_AT1K0_GAS_GPI_130.i_iPRESS_R
//     PlcTask Inputs/GVL_Devices.fb_AT1K0_GAS_GPI_140.i_iPRESS_R <-> AI Standard Channel 2/fb_AT1K0_GAS_GPI_140.i_iPRESS_R
//   plc_kfe_gatt Instance <-> =+-CX2020/EtherCAT1/=+-EK1100_02_00/=+-ES1004_02_02
//     PlcTask Inputs/GVL_Devices.fb_AT1K0_GAS_VRC_10.i_xClsLS <-> Channel 2/fb_AT1K0_GAS_VRC_10.i_xClsLS
//     PlcTask Inputs/GVL_Devices.fb_AT1K0_GAS_VRC_20.i_xClsLS <-> Channel 4/fb_AT1K0_GAS_VRC_20.i_xClsLS
//     PlcTask Inputs/GVL_Devices.fb_AT1K0_GAS_VRC_10.i_xOpnLS <-> Channel 1/fb_AT1K0_GAS_VRC_10.i_xOpnLS
//     PlcTask Inputs/GVL_Devices.fb_AT1K0_GAS_VRC_20.i_xOpnLS <-> Channel 3/fb_AT1K0_GAS_VRC_20.i_xOpnLS
//   plc_kfe_gatt Instance <-> =+-CX2020/EtherCAT1/=+-EK1100_02_00/=+-ES1004_02_04
//     PlcTask Inputs/GVL_Devices.fb_AT1K0_GAS_VRC_30.i_xClsLS <-> Channel 2/fb_AT1K0_GAS_VRC_30.i_xClsLS
//     PlcTask Inputs/GVL_Devices.fb_AT1K0_GAS_VRC_40.i_xClsLS <-> Channel 4/fb_AT1K0_GAS_VRC_40.i_xClsLS
//     PlcTask Inputs/GVL_Devices.fb_AT1K0_GAS_VRC_30.i_xOpnLS <-> Channel 1/fb_AT1K0_GAS_VRC_30.i_xOpnLS
//     PlcTask Inputs/GVL_Devices.fb_AT1K0_GAS_VRC_40.i_xOpnLS <-> Channel 3/fb_AT1K0_GAS_VRC_40.i_xOpnLS
//   plc_kfe_gatt Instance <-> =+-CX2020/EtherCAT1/=+-EK1100_02_00/=+-ES1004_02_08
//     PlcTask Inputs/GVL_Devices.fb_AT1K0_GAS_VRC_50.i_xClsLS <-> Channel 2/Input
//     PlcTask Inputs/GVL_Devices.fb_AT1K0_GAS_VRC_60.i_xClsLS <-> Channel 4/Input
//     PlcTask Inputs/GVL_Devices.fb_AT1K0_GAS_VRC_50.i_xOpnLS <-> Channel 1/Input
//     PlcTask Inputs/GVL_Devices.fb_AT1K0_GAS_VRC_60.i_xOpnLS <-> Channel 3/Input
//   plc_kfe_gatt Instance <-> =+-CX2020/EtherCAT1/=+-EK1100_02_00/=+-ES2004_02_01
//     PlcTask Outputs/GVL_Devices.fb_AT1K0_GAS_VRC_10.q_xOPN_DO <-> Channel 1/fb_AT1K0_GAS_VRC_10.q_xOPN_DO
//     PlcTask Outputs/GVL_Devices.fb_AT1K0_GAS_VRC_20.q_xOPN_DO <-> Channel 3/fb_AT1K0_GAS_VRC_20.q_xOPN_DO
//     PlcTask Outputs/GVL_Devices.fb_AT1K0_GAS_VRC_10.q_xOPN_DO_2 <-> Channel 2/fb_AT1K0_GAS_VRC_10.q_xOPN_DO
//     PlcTask Outputs/GVL_Devices.fb_AT1K0_GAS_VRC_20.q_xOPN_DO_2 <-> Channel 4/fb_AT1K0_GAS_VRC_20.q_xOPN_DO
//   plc_kfe_gatt Instance <-> =+-CX2020/EtherCAT1/=+-EK1100_02_00/=+-ES2004_02_03
//     PlcTask Outputs/GVL_Devices.fb_AT1K0_GAS_VRC_30.q_xOPN_DO <-> Channel 1/fb_AT1K0_GAS_VRC_30.q_xOPN_DO
//     PlcTask Outputs/GVL_Devices.fb_AT1K0_GAS_VRC_40.q_xOPN_DO <-> Channel 3/fb_AT1K0_GAS_VRC_40.q_xOPN_DO
//     PlcTask Outputs/GVL_Devices.fb_AT1K0_GAS_VRC_30.q_xOPN_DO_2 <-> Channel 2/fb_AT1K0_GAS_VRC_30.q_xOPN_DO
//     PlcTask Outputs/GVL_Devices.fb_AT1K0_GAS_VRC_40.q_xOPN_DO_2 <-> Channel 4/fb_AT1K0_GAS_VRC_40.q_xOPN_DO
//   plc_kfe_gatt Instance <-> =+-CX2020/EtherCAT1/=+-EK1100_02_00/=+-ES2004_02_07
//     PlcTask Outputs/GVL_Devices.fb_AT1K0_GAS_VRC_50.q_xOPN_DO <-> Channel 1/Output
//     PlcTask Outputs/GVL_Devices.fb_AT1K0_GAS_VRC_60.q_xOPN_DO <-> Channel 2/Output
//     PlcTask Outputs/Main.M2.bBrakeRelease <-> Channel 3/Output
//     PlcTask Outputs/Main.M4.bBrakeRelease <-> Channel 4/Output
//   plc_kfe_gatt Instance <-> =+-CX2020/EtherCAT1/=+-EK1100_02_00/=+-ES7041_02_05
//     PlcTask Inputs/Main.M1.bLimitBackwardEnable <-> STM Status/Status/Digital input 2
//     PlcTask Inputs/Main.M1.bLimitForwardEnable <-> STM Status/Status/Digital input 1
//   plc_kfe_gatt Instance <-> =+-CX2020/EtherCAT1/=+-EK1100_02_00/=+-ES7041_02_06
//     PlcTask Inputs/Main.M2.bLimitBackwardEnable <-> STM Status/Status/Digital input 1
//     PlcTask Inputs/Main.M2.bLimitForwardEnable <-> STM Status/Status/Digital input 2
//   plc_kfe_gatt Instance <-> =+-CX2020/EtherCAT1/=+-EK1100_02_00/=+-ES7041_02_09
//     PlcTask Inputs/Main.M3.bLimitBackwardEnable <-> STM Status/Status/Digital input 2
//     PlcTask Inputs/Main.M3.bLimitForwardEnable <-> STM Status/Status/Digital input 1
//   plc_kfe_gatt Instance <-> =+-CX2020/EtherCAT1/=+-EK1100_02_00/=+-ES7041_02_10
//     PlcTask Inputs/Main.M4.bLimitBackwardEnable <-> STM Status/Status/Digital input 1
//     PlcTask Inputs/Main.M4.bLimitForwardEnable <-> STM Status/Status/Digital input 2
//   plc_kfe_gatt Instance <-> =+-CX2020/EtherCAT1/=+-EK1100_03_00/=+-EL2798_03_03
//     PlcTask Outputs/GVL_Devices.fb_AT1K0_GAS_PTM_10.q_xProtection <-> Channel 4/fb_AT1K0_GAS_PTM_10.q_xProtection
//     PlcTask Outputs/GVL_Devices.fb_AT1K0_GAS_PTM_10.q_xReset <-> Channel 1/fb_AT1K0_GAS_PTM_10.q_xReset
//     PlcTask Outputs/GVL_Devices.fb_AT1K0_GAS_PTM_10.q_xSetSpeed <-> Channel 5/fb_AT1K0_GAS_PTM_10.q_xSetSpeed
//     PlcTask Outputs/GVL_Devices.fb_AT1K0_GAS_PTM_10.q_xStart <-> Channel 2/fb_AT1K0_GAS_PTM_10.q_xStart
//     PlcTask Outputs/GVL_Devices.fb_AT1K0_GAS_PTM_10.q_xStop <-> Channel 3/fb_AT1K0_GAS_PTM_10.q_xStop
//   plc_kfe_gatt Instance <-> =+-CX2020/EtherCAT1/=+-EK1100_03_00/=+-EL2798_03_07
//     PlcTask Outputs/GVL_Devices.fb_AT1K0_GAS_PTM_20.q_xProtection <-> Channel 4/fb_AT1K0_GAS_PTM_20.q_xProtection
//     PlcTask Outputs/GVL_Devices.fb_AT1K0_GAS_PTM_20.q_xReset <-> Channel 1/fb_AT1K0_GAS_PTM_20.q_xReset
//     PlcTask Outputs/GVL_Devices.fb_AT1K0_GAS_PTM_20.q_xSetSpeed <-> Channel 5/fb_AT1K0_GAS_PTM_20.q_xSetSpeed
//     PlcTask Outputs/GVL_Devices.fb_AT1K0_GAS_PTM_20.q_xStart <-> Channel 2/fb_AT1K0_GAS_PTM_20.q_xStart
//     PlcTask Outputs/GVL_Devices.fb_AT1K0_GAS_PTM_20.q_xStop <-> Channel 3/fb_AT1K0_GAS_PTM_20.q_xStop
//   plc_kfe_gatt Instance <-> =+-CX2020/EtherCAT1/=+-EK1100_03_00/=+-EL2798_03_13
//     PlcTask Outputs/GVL_Devices.fb_AT1K0_GAS_PTM_30.q_xProtection <-> Channel 4/fb_AT1K0_GAS_PTM_30.q_xProtection
//     PlcTask Outputs/GVL_Devices.fb_AT1K0_GAS_PTM_30.q_xReset <-> Channel 1/fb_AT1K0_GAS_PTM_30.q_xReset
//     PlcTask Outputs/GVL_Devices.fb_AT1K0_GAS_PTM_30.q_xSetSpeed <-> Channel 5/fb_AT1K0_GAS_PTM_30.q_xSetSpeed
//     PlcTask Outputs/GVL_Devices.fb_AT1K0_GAS_PTM_30.q_xStart <-> Channel 2/fb_AT1K0_GAS_PTM_30.q_xStart
//     PlcTask Outputs/GVL_Devices.fb_AT1K0_GAS_PTM_30.q_xStop <-> Channel 3/fb_AT1K0_GAS_PTM_30.q_xStop
//   plc_kfe_gatt Instance <-> =+-CX2020/EtherCAT1/=+-EK1100_03_00/=+-EL2798_03_17
//     PlcTask Outputs/GVL_Devices.fb_AT1K0_GAS_PTM_40.q_xProtection <-> Channel 4/fb_AT1K0_GAS_PTM_40.q_xProtection
//     PlcTask Outputs/GVL_Devices.fb_AT1K0_GAS_PTM_40.q_xReset <-> Channel 1/fb_AT1K0_GAS_PTM_40.q_xReset
//     PlcTask Outputs/GVL_Devices.fb_AT1K0_GAS_PTM_40.q_xSetSpeed <-> Channel 5/fb_AT1K0_GAS_PTM_40.q_xSetSpeed
//     PlcTask Outputs/GVL_Devices.fb_AT1K0_GAS_PTM_40.q_xStart <-> Channel 2/fb_AT1K0_GAS_PTM_40.q_xStart
//     PlcTask Outputs/GVL_Devices.fb_AT1K0_GAS_PTM_40.q_xStop <-> Channel 3/fb_AT1K0_GAS_PTM_40.q_xStop
//   plc_kfe_gatt Instance <-> =+-CX2020/EtherCAT1/=+-EK1100_03_00/=+-ES1004_03_01
//     PlcTask Inputs/GVL_Devices.fb_AT1K0_GAS_PTM_10.i_xAtSpd <-> Channel 2/fb_AT1K0_GAS_PTM_10.i_xAtSpd
//     PlcTask Inputs/GVL_Devices.fb_AT1K0_GAS_PTM_10.i_xDecel <-> Channel 1/fb_AT1K0_GAS_PTM_10.i_xDecel
//     PlcTask Inputs/GVL_Devices.fb_AT1K0_GAS_PTM_10.i_xNCFault <-> Channel 3/fb_AT1K0_GAS_PTM_10.i_xNCFault
//     PlcTask Inputs/GVL_Devices.fb_AT1K0_GAS_PTM_10.i_xRotate <-> Channel 4/fb_AT1K0_GAS_PTM_10.i_xRotate
//   plc_kfe_gatt Instance <-> =+-CX2020/EtherCAT1/=+-EK1100_03_00/=+-ES1004_03_02
//     PlcTask Inputs/GVL_Devices.fb_AT1K0_GAS_PTM_10.i_xAccel <-> Channel 1/fb_AT1K0_GAS_PTM_10.i_xAccel
//   plc_kfe_gatt Instance <-> =+-CX2020/EtherCAT1/=+-EK1100_03_00/=+-ES1004_03_08
//     PlcTask Inputs/GVL_Devices.fb_AT1K0_GAS_PTM_20.i_xAtSpd <-> Channel 2/fb_AT1K0_GAS_PTM_20.i_xAtSpd
//     PlcTask Inputs/GVL_Devices.fb_AT1K0_GAS_PTM_20.i_xDecel <-> Channel 1/fb_AT1K0_GAS_PTM_20.i_xDecel
//     PlcTask Inputs/GVL_Devices.fb_AT1K0_GAS_PTM_20.i_xNCFault <-> Channel 3/fb_AT1K0_GAS_PTM_20.i_xNCFault
//     PlcTask Inputs/GVL_Devices.fb_AT1K0_GAS_PTM_20.i_xRotate <-> Channel 4/fb_AT1K0_GAS_PTM_20.i_xRotate
//   plc_kfe_gatt Instance <-> =+-CX2020/EtherCAT1/=+-EK1100_03_00/=+-ES1004_03_09
//     PlcTask Inputs/GVL_Devices.fb_AT1K0_GAS_PTM_20.i_xAccel <-> Channel 1/fb_AT1K0_GAS_PTM_20.i_xAccel
//   plc_kfe_gatt Instance <-> =+-CX2020/EtherCAT1/=+-EK1100_03_00/=+-ES1004_03_11
//     PlcTask Inputs/GVL_Devices.fb_AT1K0_GAS_PTM_30.i_xAtSpd <-> Channel 2/fb_AT1K0_GAS_PTM_30.i_xAtSpd
//     PlcTask Inputs/GVL_Devices.fb_AT1K0_GAS_PTM_30.i_xDecel <-> Channel 1/fb_AT1K0_GAS_PTM_30.i_xDecel
//     PlcTask Inputs/GVL_Devices.fb_AT1K0_GAS_PTM_30.i_xNCFault <-> Channel 3/fb_AT1K0_GAS_PTM_30.i_xNCFault
//     PlcTask Inputs/GVL_Devices.fb_AT1K0_GAS_PTM_30.i_xRotate <-> Channel 4/fb_AT1K0_GAS_PTM_30.i_xRotate
//   plc_kfe_gatt Instance <-> =+-CX2020/EtherCAT1/=+-EK1100_03_00/=+-ES1004_03_12
//     PlcTask Inputs/GVL_Devices.fb_AT1K0_GAS_PTM_30.i_xAccel <-> Channel 1/fb_AT1K0_GAS_PTM_30.i_xAccel
//   plc_kfe_gatt Instance <-> =+-CX2020/EtherCAT1/=+-EK1100_03_00/=+-ES1004_03_18
//     PlcTask Inputs/GVL_Devices.fb_AT1K0_GAS_PTM_40.i_xAtSpd <-> Channel 2/fb_AT1K0_GAS_PTM_40.i_xAtSpd
//     PlcTask Inputs/GVL_Devices.fb_AT1K0_GAS_PTM_40.i_xDecel <-> Channel 1/fb_AT1K0_GAS_PTM_40.i_xDecel
//     PlcTask Inputs/GVL_Devices.fb_AT1K0_GAS_PTM_40.i_xNCFault <-> Channel 3/fb_AT1K0_GAS_PTM_40.i_xNCFault
//     PlcTask Inputs/GVL_Devices.fb_AT1K0_GAS_PTM_40.i_xRotate <-> Channel 4/fb_AT1K0_GAS_PTM_40.i_xRotate
//   plc_kfe_gatt Instance <-> =+-CX2020/EtherCAT1/=+-EK1100_03_00/=+-ES1004_03_19
//     PlcTask Inputs/GVL_Devices.fb_AT1K0_GAS_PTM_40.i_xAccel <-> Channel 1/fb_AT1K0_GAS_PTM_40.i_xAccel
//   plc_kfe_gatt Instance <-> =+-CX2020/EtherCAT1/=+-EK1100_03_00/=+-ES3064_03_04
//     PlcTask Inputs/GVL_Devices.fb_AT1K0_GAS_PTM_10.i_iCurrentMon <-> AI Standard Channel 2/fb_AT1K0_GAS_PTM_10.i_iCurrentMon
//     PlcTask Inputs/GVL_Devices.fb_AT1K0_GAS_PTM_10.i_iRawSpeed <-> AI Standard Channel 1/fb_AT1K0_GAS_PTM_10.i_iRawSpeed
//     PlcTask Inputs/GVL_Devices.fb_AT1K0_GAS_PTM_10.i_iTempMon <-> AI Standard Channel 3/fb_AT1K0_GAS_PTM_10.i_iTempMon
//   plc_kfe_gatt Instance <-> =+-CX2020/EtherCAT1/=+-EK1100_03_00/=+-ES3064_03_06
//     PlcTask Inputs/GVL_Devices.fb_AT1K0_GAS_PTM_20.i_iCurrentMon <-> AI Standard Channel 2/fb_AT1K0_GAS_PTM_20.i_iCurrentMon
//     PlcTask Inputs/GVL_Devices.fb_AT1K0_GAS_PTM_20.i_iRawSpeed <-> AI Standard Channel 1/fb_AT1K0_GAS_PTM_20.i_iRawSpeed
//     PlcTask Inputs/GVL_Devices.fb_AT1K0_GAS_PTM_20.i_iTempMon <-> AI Standard Channel 3/fb_AT1K0_GAS_PTM_20.i_iTempMon
//   plc_kfe_gatt Instance <-> =+-CX2020/EtherCAT1/=+-EK1100_03_00/=+-ES3064_03_14
//     PlcTask Inputs/GVL_Devices.fb_AT1K0_GAS_PTM_30.i_iCurrentMon <-> AI Standard Channel 2/fb_AT1K0_GAS_PTM_30.i_iCurrentMon
//     PlcTask Inputs/GVL_Devices.fb_AT1K0_GAS_PTM_30.i_iRawSpeed <-> AI Standard Channel 1/fb_AT1K0_GAS_PTM_30.i_iRawSpeed
//     PlcTask Inputs/GVL_Devices.fb_AT1K0_GAS_PTM_30.i_iTempMon <-> AI Standard Channel 3/fb_AT1K0_GAS_PTM_30.i_iTempMon
//   plc_kfe_gatt Instance <-> =+-CX2020/EtherCAT1/=+-EK1100_03_00/=+-ES3064_03_16
//     PlcTask Inputs/GVL_Devices.fb_AT1K0_GAS_PTM_40.i_iCurrentMon <-> AI Standard Channel 2/fb_AT1K0_GAS_PTM_40.i_iCurrentMon
//     PlcTask Inputs/GVL_Devices.fb_AT1K0_GAS_PTM_40.i_iRawSpeed <-> AI Standard Channel 1/fb_AT1K0_GAS_PTM_40.i_iRawSpeed
//     PlcTask Inputs/GVL_Devices.fb_AT1K0_GAS_PTM_40.i_iTempMon <-> AI Standard Channel 3/fb_AT1K0_GAS_PTM_40.i_iTempMon
//   plc_kfe_gatt Instance <-> =+-CX2020/EtherCAT1/=+-EK1100_03_00/=+-ES4004_03_05
//     PlcTask Outputs/GVL_Devices.fb_AT1K0_GAS_PTM_10.q_iSpeedSet <-> AO Outputs Channel 1/fb_AT1K0_GAS_PTM_10.q_iSpeedSet
//     PlcTask Outputs/GVL_Devices.fb_AT1K0_GAS_PTM_20.q_iSpeedSet <-> AO Outputs Channel 3/fb_AT1K0_GAS_PTM_20.q_iSpeedSet
//   plc_kfe_gatt Instance <-> =+-CX2020/EtherCAT1/=+-EK1100_03_00/=+-ES4004_03_15
//     PlcTask Outputs/GVL_Devices.fb_AT1K0_GAS_PTM_30.q_iSpeedSet <-> AO Outputs Channel 1/fb_AT1K0_GAS_PTM_30.q_iSpeedSet
//     PlcTask Outputs/GVL_Devices.fb_AT1K0_GAS_PTM_40.q_iSpeedSet <-> AO Outputs Channel 3/fb_AT1K0_GAS_PTM_40.q_iSpeedSet
//   plc_kfe_gatt Instance <-> =+-CX2020/EtherCAT1/=+-EK1100_04_00/=+-EL3174_04_17
//     PlcTask Inputs/GVL_Devices.GCM_70.i_iPRESS_R <-> AI Standard Channel 3/GCM_70.i_iPRESS_R
//     PlcTask Inputs/GVL_Devices.GCM_80.i_iPRESS_R <-> AI Standard Channel 1/GCM_80.i_iPRESS_R
//     PlcTask Inputs/GVL_Devices.GCM_81.i_iPRESS_R <-> AI Standard Channel 2/Value
//   plc_kfe_gatt Instance <-> =+-CX2020/EtherCAT1/=+-EK1100_04_00/=+-EL7041_04_07
//     PlcTask Inputs/Main.M5.bLimitBackwardEnable <-> STM Status/Status/Digital input 1
//     PlcTask Inputs/Main.M5.bLimitForwardEnable <-> STM Status/Status/Digital input 2
//   plc_kfe_gatt Instance <-> =+-CX2020/EtherCAT1/=+-EK1100_04_00/=+-EL7041_04_08
//     PlcTask Inputs/Main.M6.bLimitBackwardEnable <-> STM Status/Status/Digital input 1
//     PlcTask Inputs/Main.M6.bLimitForwardEnable <-> STM Status/Status/Digital input 2
//   plc_kfe_gatt Instance <-> =+-CX2020/EtherCAT1/=+-EK1100_04_00/=+-EL7041_04_10
//     PlcTask Inputs/Main.M7.bLimitBackwardEnable <-> STM Status/Status/Digital input 1
//     PlcTask Inputs/Main.M7.bLimitForwardEnable <-> STM Status/Status/Digital input 2
//   plc_kfe_gatt Instance <-> =+-CX2020/EtherCAT1/=+-EK1100_04_00/=+-EL7041_04_11
//     PlcTask Inputs/Main.M8.bLimitBackwardEnable <-> STM Status/Status/Digital input 1
//     PlcTask Inputs/Main.M8.bLimitForwardEnable <-> STM Status/Status/Digital input 2
//   plc_kfe_gatt Instance <-> =+-CX2020/EtherCAT1/=+-EK1100_04_00/=+-ES1084_04_06
//     PlcTask Inputs/GVL_Devices.fb_AT1K0_GAS_PTM_80.i_xAtSpd <-> Channel 1/fb_AT1K0_GAS_PTM_80.i_xAtSpd
//     PlcTask Inputs/GVL_Devices.fb_AT1K0_GAS_PTM_80.i_xFault <-> Channel 2/fb_AT1K0_GAS_PTM_80.i_xFault
//   plc_kfe_gatt Instance <-> =+-CX2020/EtherCAT1/=+-EK1100_04_00/=+-ES2004_04_01
//     PlcTask Outputs/GVL_Devices.VVC_71.q_xOPN_DO <-> Channel 1/VVC_71.q_xOPN_DO
//     PlcTask Outputs/GVL_Devices.VVC_72.q_xOPN_DO <-> Channel 2/VVC_72.q_xOPN_DO
//     PlcTask Outputs/GVL_Devices.fb_AT1K0_GAS_PTM_80.q_RunDO <-> Channel 3/fb_AT1K0_GAS_PTM_80.q_RunDO
//   plc_kfe_gatt Instance <-> =+-CX2020/EtherCAT1/=+-EK1100_04_00/=+-ES2004_04_09
//     PlcTask Outputs/Main.M{5..8}.bBrakeRelease <-> Channel {1..4}/Output  (4 links)
//   plc_kfe_gatt Instance <-> =+-CX2020/EtherCAT1/=+-EK1100_04_00/=+-ES4004_04_02
//     PlcTask Outputs/GVL_Devices.VCN_70.q_iRawPosition <-> AO Outputs Channel 1/VCN_70.q_iRawPosition
//   plc_kfe_gatt Instance <-> =+-CX2020/EtherCAT1/=+-EK1100_05_00/=+-EL1084_05_12
//     PlcTask Inputs/GVL_Devices.fb_AT1K0_GAS_PMF_110.i_xAlarmOK <-> Channel 2/fb_AT1K0_GAS_PMF_110.i_xAlarmOK
//     PlcTask Inputs/GVL_Devices.fb_AT1K0_GAS_PMF_120.i_xAlarmOK <-> Channel 4/fb_AT1K0_GAS_PMF_120.i_xAlarmOK
//     PlcTask Inputs/GVL_Devices.fb_AT1K0_GAS_PMF_110.i_xIsRun <-> Channel 1/fb_AT1K0_GAS_PMF_110.i_xIsRun
//     PlcTask Inputs/GVL_Devices.fb_AT1K0_GAS_PMF_120.i_xIsRun <-> Channel 3/fb_AT1K0_GAS_PMF_120.i_xIsRun
//   plc_kfe_gatt Instance <-> =+-CX2020/EtherCAT1/=+-EK1100_05_00/=+-EL1084_05_13
//     PlcTask Inputs/GVL_Devices.fb_AT1K0_GAS_PMF_140.i_xAlarmOK <-> Channel 2/fb_AT1K0_GAS_PMF_140.i_xAlarmOK
//     PlcTask Inputs/GVL_Devices.fb_AT1K0_GAS_PMF_140.i_xIsRun <-> Channel 1/fb_AT1K0_GAS_PMF_140.i_xIsRun
//   plc_kfe_gatt Instance <-> =+-CX2020/EtherCAT1/=+-EK1100_05_00/=+-EL2798_05_10
//     PlcTask Outputs/GVL_Devices.fb_AT1K0_GAS_PMF_110.q_xResetAlarm <-> Channel 2/fb_AT1K0_GAS_PMF_110.q_xResetAlarm
//     PlcTask Outputs/GVL_Devices.fb_AT1K0_GAS_PMF_120.q_xResetAlarm <-> Channel 4/fb_AT1K0_GAS_PMF_120.q_xResetAlarm
//     PlcTask Outputs/GVL_Devices.fb_AT1K0_GAS_PMF_140.q_xResetAlarm <-> Channel 6/fb_AT1K0_GAS_PMF_140.q_xResetAlarm
//     PlcTask Outputs/GVL_Devices.fb_AT1K0_GAS_PMF_110.q_xRunDo <-> Channel 1/fb_AT1K0_GAS_PMF_110.q_xRunDo
//     PlcTask Outputs/GVL_Devices.fb_AT1K0_GAS_PMF_120.q_xRunDo <-> Channel 3/fb_AT1K0_GAS_PMF_120.q_xRunDo
//     PlcTask Outputs/GVL_Devices.fb_AT1K0_GAS_PMF_140.q_xRunDo <-> Channel 5/fb_AT1K0_GAS_PMF_140.q_xRunDo
//   plc_kfe_gatt Instance <-> =+-CX2020/EtherCAT1/=+-EK1100_05_00/=+-EL3174_05_16
//     PlcTask Inputs/GVL_Devices.fb_AT1K0_GAS_GPI_111.i_iPRESS_R <-> AI Standard Channel 1/fb_AT1K0_GAS_GPI_111.i_iPRESS_R
//     PlcTask Inputs/GVL_Devices.fb_AT1K0_GAS_GPI_141.i_iPRESS_R <-> AI Standard Channel 3/fb_AT1K0_GAS_GPI_141.i_iPRESS_R
//     PlcTask Inputs/GVL_Devices.fb_AT1K0_GAS_GPI_121.i_iPRESS_R <-> AI Standard Channel 2/Value
//   plc_kfe_gatt Instance <-> =+-CX2020/EtherCAT1/=+-EK1100_05_00/=+-ES1004_05_01
//     PlcTask Inputs/GVL_Devices.fb_AT1K0_GAS_VRC_70.i_xClsLS <-> Channel 2/fb_AT1K0_GAS_VRC_70.i_xClsLS
//     PlcTask Inputs/GVL_Devices.fb_AT1K0_GAS_VRC_80.i_xClsLS <-> Channel 4/fb_AT1K0_GAS_VRC_80.i_xClsLS
//     PlcTask Inputs/GVL_Devices.fb_AT1K0_GAS_VRC_70.i_xOpnLS <-> Channel 1/fb_AT1K0_GAS_VRC_70.i_xOpnLS
//     PlcTask Inputs/GVL_Devices.fb_AT1K0_GAS_VRC_80.i_xOpnLS <-> Channel 3/fb_AT1K0_GAS_VRC_80.i_xOpnLS
//   plc_kfe_gatt Instance <-> =+-CX2020/EtherCAT1/=+-EK1100_05_00/=+-ES1004_05_03
//     PlcTask Inputs/GVL_Devices.fb_AT1K0_GAS_VRC_100.i_xClsLS <-> Channel 4/fb_AT1K0_GAS_VRC_100.i_xClsLS
//     PlcTask Inputs/GVL_Devices.fb_AT1K0_GAS_VRC_90.i_xClsLS <-> Channel 2/fb_AT1K0_GAS_VRC_90.i_xClsLS
//     PlcTask Inputs/GVL_Devices.fb_AT1K0_GAS_VRC_100.i_xOpnLS <-> Channel 3/fb_AT1K0_GAS_VRC_100.i_xOpnLS
//     PlcTask Inputs/GVL_Devices.fb_AT1K0_GAS_VRC_90.i_xOpnLS <-> Channel 1/fb_AT1K0_GAS_VRC_90.i_xOpnLS
//   plc_kfe_gatt Instance <-> =+-CX2020/EtherCAT1/=+-EK1100_05_00/=+-ES1004_05_06
//     PlcTask Inputs/GVL_Devices.fb_AT1K0_GAS_VRC_110.i_xClsLS <-> Channel 2/fb_AT1K0_GAS_VRC_110.i_xClsLS
//     PlcTask Inputs/GVL_Devices.fb_AT1K0_GAS_VRC_120.i_xClsLS <-> Channel 4/fb_AT1K0_GAS_VRC_120.i_xClsLS
//     PlcTask Inputs/GVL_Devices.fb_AT1K0_GAS_VRC_110.i_xOpnLS <-> Channel 1/fb_AT1K0_GAS_VRC_110.i_xOpnLS
//     PlcTask Inputs/GVL_Devices.fb_AT1K0_GAS_VRC_120.i_xOpnLS <-> Channel 3/fb_AT1K0_GAS_VRC_120.i_xOpnLS
//   plc_kfe_gatt Instance <-> =+-CX2020/EtherCAT1/=+-EK1100_05_00/=+-ES1004_05_08
//     PlcTask Inputs/GVL_Devices.fb_AT1K0_GAS_VRC_130.i_xClsLS <-> Channel 2/fb_AT1K0_GAS_VRC_130.i_xClsLS
//     PlcTask Inputs/GVL_Devices.fb_AT1K0_GAS_VRC_140.i_xClsLS <-> Channel 4/fb_AT1K0_GAS_VRC_140.i_xClsLS
//     PlcTask Inputs/GVL_Devices.fb_AT1K0_GAS_VRC_130.i_xOpnLS <-> Channel 1/fb_AT1K0_GAS_VRC_130.i_xOpnLS
//     PlcTask Inputs/GVL_Devices.fb_AT1K0_GAS_VRC_140.i_xOpnLS <-> Channel 3/fb_AT1K0_GAS_VRC_140.i_xOpnLS
//   plc_kfe_gatt Instance <-> =+-CX2020/EtherCAT1/=+-EK1100_05_00/=+-ES2004_05_02
//     PlcTask Outputs/GVL_Devices.fb_AT1K0_GAS_VRC_70.q_xOPN_DO <-> Channel 1/fb_AT1K0_GAS_VRC_70.q_xOPN_DO
//     PlcTask Outputs/GVL_Devices.fb_AT1K0_GAS_VRC_80.q_xOPN_DO <-> Channel 2/fb_AT1K0_GAS_VRC_80.q_xOPN_DO
//   plc_kfe_gatt Instance <-> =+-CX2020/EtherCAT1/=+-EK1100_05_00/=+-ES2004_05_04
//     PlcTask Outputs/GVL_Devices.fb_AT1K0_GAS_VRC_100.q_xOPN_DO <-> Channel 2/fb_AT1K0_GAS_VRC_100.q_xOPN_DO
//     PlcTask Outputs/GVL_Devices.fb_AT1K0_GAS_VRC_90.q_xOPN_DO <-> Channel 1/fb_AT1K0_GAS_VRC_90.q_xOPN_DO
//   plc_kfe_gatt Instance <-> =+-CX2020/EtherCAT1/=+-EK1100_05_00/=+-ES2004_05_05
//     PlcTask Outputs/GVL_Devices.fb_AT1K0_GAS_VRC_110.q_xOPN_DO <-> Channel 1/fb_AT1K0_GAS_VRC_110.q_xOPN_DO
//     PlcTask Outputs/GVL_Devices.fb_AT1K0_GAS_VRC_120.q_xOPN_DO <-> Channel 2/fb_AT1K0_GAS_VRC_120.q_xOPN_DO
//   plc_kfe_gatt Instance <-> =+-CX2020/EtherCAT1/=+-EK1100_05_00/=+-ES2004_05_07
//     PlcTask Outputs/GVL_Devices.fb_AT1K0_GAS_VRC_130.q_xOPN_DO <-> Channel 1/fb_AT1K0_GAS_VRC_130.q_xOPN_DO
//     PlcTask Outputs/GVL_Devices.fb_AT1K0_GAS_VRC_140.q_xOPN_DO <-> Channel 2/fb_AT1K0_GAS_VRC_140.q_xOPN_DO
//   plc_kfe_gatt Instance <-> =+-CX2020/EtherCAT1/=+-EK1100_06_00/=+-EL2212_06_25
//     PlcTask Outputs/GVL_Devices.fb_AT1K0_GAS_VVC_110.q_xOPN_DO <-> DOX Control Channel 1/Control/Output
//     PlcTask Outputs/GVL_Devices.fb_AT1K0_GAS_VVC_120.q_xOPN_DO <-> DOX Control Channel 2/Control/Output
//   plc_kfe_gatt Instance <-> =+-CX2020/EtherCAT1/=+-EK1100_06_00/=+-EL2212_06_26
//     PlcTask Outputs/GVL_Devices.fb_AT1K0_GAS_VVC_140.q_xOPN_DO <-> DOX Control Channel 1/Control/Output
//     PlcTask Outputs/GVL_Devices.fb_AT1K0_GAS_VVC_80.q_xOPN_DO <-> DOX Control Channel 2/Control/Output
//   plc_kfe_gatt Instance <-> =+-CX2020/EtherCAT1/=+-EK1100_06_00/=+-EL2794_06_22
//     PlcTask Outputs/GVL_Devices.fb_AT1K0_GAS_PMF_100.q_xBPStart <-> Channel 4/fb_AT1K0_GAS_PMF_100.q_xBPStart
//     PlcTask Outputs/GVL_Devices.fb_AT1K0_GAS_PMF_90.q_xBPStart <-> Channel 2/fb_AT1K0_GAS_PMF_90.q_xBPStart
//     PlcTask Outputs/GVL_Devices.fb_AT1K0_GAS_PMF_100.q_xMPStart <-> Channel 3/fb_AT1K0_GAS_PMF_100.q_xMPStart
//     PlcTask Outputs/GVL_Devices.fb_AT1K0_GAS_PMF_90.q_xMPStart <-> Channel 1/fb_AT1K0_GAS_PMF_90.q_xMPStart
//   plc_kfe_gatt Instance <-> =+-CX2020/EtherCAT1/=+-EK1100_06_00/=+-EL2798_06_03
//     PlcTask Outputs/GVL_Devices.fb_AT1K0_GAS_PTM_110.q_xProtection <-> Channel 5/fb_AT1K0_GAS_PTM_110.q_xProtection
//     PlcTask Outputs/GVL_Devices.fb_AT1K0_GAS_PTM_110.q_xReset <-> Channel 1/fb_AT1K0_GAS_PTM_110.q_xReset
//     PlcTask Outputs/GVL_Devices.fb_AT1K0_GAS_PTM_110.q_xSetSpeed <-> Channel 4/fb_AT1K0_GAS_PTM_110.q_xSetSpeed
//     PlcTask Outputs/GVL_Devices.fb_AT1K0_GAS_PTM_110.q_xStart <-> Channel 2/fb_AT1K0_GAS_PTM_110.q_xStart
//     PlcTask Outputs/GVL_Devices.fb_AT1K0_GAS_PTM_110.q_xStop <-> Channel 3/fb_AT1K0_GAS_PTM_110.q_xStop
//   plc_kfe_gatt Instance <-> =+-CX2020/EtherCAT1/=+-EK1100_06_00/=+-EL2798_06_07
//     PlcTask Outputs/GVL_Devices.fb_AT1K0_GAS_PTM_120.q_xProtection <-> Channel 4/fb_AT1K0_GAS_PTM_120.q_xProtection
//     PlcTask Outputs/GVL_Devices.fb_AT1K0_GAS_PTM_120.q_xReset <-> Channel 1/fb_AT1K0_GAS_PTM_120.q_xReset
//     PlcTask Outputs/GVL_Devices.fb_AT1K0_GAS_PTM_120.q_xSetSpeed <-> Channel 5/fb_AT1K0_GAS_PTM_120.q_xSetSpeed
//     PlcTask Outputs/GVL_Devices.fb_AT1K0_GAS_PTM_120.q_xStart <-> Channel 2/fb_AT1K0_GAS_PTM_120.q_xStart
//     PlcTask Outputs/GVL_Devices.fb_AT1K0_GAS_PTM_120.q_xStop <-> Channel 3/fb_AT1K0_GAS_PTM_120.q_xStop
//   plc_kfe_gatt Instance <-> =+-CX2020/EtherCAT1/=+-EK1100_06_00/=+-EL2798_06_13
//     PlcTask Outputs/GVL_Devices.fb_AT1K0_GAS_PTM_130.q_xProtection <-> Channel 4/fb_AT1K0_GAS_PTM_130.q_xProtection
//     PlcTask Outputs/GVL_Devices.fb_AT1K0_GAS_PTM_130.q_xReset <-> Channel 1/fb_AT1K0_GAS_PTM_130.q_xReset
//     PlcTask Outputs/GVL_Devices.fb_AT1K0_GAS_PTM_130.q_xSetSpeed <-> Channel 5/fb_AT1K0_GAS_PTM_130.q_xSetSpeed
//     PlcTask Outputs/GVL_Devices.fb_AT1K0_GAS_PTM_130.q_xStart <-> Channel 2/fb_AT1K0_GAS_PTM_130.q_xStart
//     PlcTask Outputs/GVL_Devices.fb_AT1K0_GAS_PTM_130.q_xStop <-> Channel 3/fb_AT1K0_GAS_PTM_130.q_xStop
//   plc_kfe_gatt Instance <-> =+-CX2020/EtherCAT1/=+-EK1100_06_00/=+-EL2798_06_17
//     PlcTask Outputs/GVL_Devices.fb_AT1K0_GAS_PTM_140.q_xProtection <-> Channel 4/fb_AT1K0_GAS_PTM_140.q_xProtection
//     PlcTask Outputs/GVL_Devices.fb_AT1K0_GAS_PTM_140.q_xReset <-> Channel 1/fb_AT1K0_GAS_PTM_140.q_xReset
//     PlcTask Outputs/GVL_Devices.fb_AT1K0_GAS_PTM_140.q_xSetSpeed <-> Channel 5/fb_AT1K0_GAS_PTM_140.q_xSetSpeed
//     PlcTask Outputs/GVL_Devices.fb_AT1K0_GAS_PTM_140.q_xStart <-> Channel 2/fb_AT1K0_GAS_PTM_140.q_xStart
//     PlcTask Outputs/GVL_Devices.fb_AT1K0_GAS_PTM_140.q_xStop <-> Channel 3/fb_AT1K0_GAS_PTM_140.q_xStop
//   plc_kfe_gatt Instance <-> =+-CX2020/EtherCAT1/=+-EK1100_06_00/=+-ES1004_06_01
//     PlcTask Inputs/GVL_Devices.fb_AT1K0_GAS_PTM_110.i_xAccel <-> Channel 4/fb_AT1K0_GAS_PTM_110.i_xAccel
//     PlcTask Inputs/GVL_Devices.fb_AT1K0_GAS_PTM_110.i_xAtSpd <-> Channel 1/fb_AT1K0_GAS_PTM_110.i_xAtSpd
//     PlcTask Inputs/GVL_Devices.fb_AT1K0_GAS_PTM_110.i_xFaultNC <-> Channel 2/fb_AT1K0_GAS_PTM_110.i_xFaultNC
//     PlcTask Inputs/GVL_Devices.fb_AT1K0_GAS_PTM_110.i_xRotate <-> Channel 3/fb_AT1K0_GAS_PTM_110.i_xRotate
//   plc_kfe_gatt Instance <-> =+-CX2020/EtherCAT1/=+-EK1100_06_00/=+-ES1004_06_02
//     PlcTask Inputs/GVL_Devices.fb_AT1K0_GAS_PTM_110.i_xDecel <-> Channel 1/fb_AT1K0_GAS_PTM_110.i_xDecel
//   plc_kfe_gatt Instance <-> =+-CX2020/EtherCAT1/=+-EK1100_06_00/=+-ES1004_06_08
//     PlcTask Inputs/GVL_Devices.fb_AT1K0_GAS_PTM_120.i_xAtSpd <-> Channel 2/fb_AT1K0_GAS_PTM_120.i_xAtSpd
//     PlcTask Inputs/GVL_Devices.fb_AT1K0_GAS_PTM_120.i_xDecel <-> Channel 1/fb_AT1K0_GAS_PTM_120.i_xDecel
//     PlcTask Inputs/GVL_Devices.fb_AT1K0_GAS_PTM_120.i_xNCFault <-> Channel 3/fb_AT1K0_GAS_PTM_120.i_xNCFault
//     PlcTask Inputs/GVL_Devices.fb_AT1K0_GAS_PTM_120.i_xRotate <-> Channel 4/fb_AT1K0_GAS_PTM_120.i_xRotate
//   plc_kfe_gatt Instance <-> =+-CX2020/EtherCAT1/=+-EK1100_06_00/=+-ES1004_06_09
//     PlcTask Inputs/GVL_Devices.fb_AT1K0_GAS_PTM_120.i_xAccel <-> Channel 1/fb_AT1K0_GAS_PTM_120.i_xAccel
//   plc_kfe_gatt Instance <-> =+-CX2020/EtherCAT1/=+-EK1100_06_00/=+-ES1004_06_11
//     PlcTask Inputs/GVL_Devices.fb_AT1K0_GAS_PTM_130.i_xAtSpd <-> Channel 2/fb_AT1K0_GAS_PTM_130.i_xAtSpd
//     PlcTask Inputs/GVL_Devices.fb_AT1K0_GAS_PTM_130.i_xDecel <-> Channel 1/fb_AT1K0_GAS_PTM_130.i_xDecel
//     PlcTask Inputs/GVL_Devices.fb_AT1K0_GAS_PTM_130.i_xNCFault <-> Channel 3/fb_AT1K0_GAS_PTM_130.i_xNCFault
//     PlcTask Inputs/GVL_Devices.fb_AT1K0_GAS_PTM_130.i_xRotate <-> Channel 4/fb_AT1K0_GAS_PTM_130.i_xRotate
//   plc_kfe_gatt Instance <-> =+-CX2020/EtherCAT1/=+-EK1100_06_00/=+-ES1004_06_12
//     PlcTask Inputs/GVL_Devices.fb_AT1K0_GAS_PTM_130.i_xAccel <-> Channel 1/fb_AT1K0_GAS_PTM_130.i_xAccel
//   plc_kfe_gatt Instance <-> =+-CX2020/EtherCAT1/=+-EK1100_06_00/=+-ES1004_06_18
//     PlcTask Inputs/GVL_Devices.fb_AT1K0_GAS_PTM_140.i_xAtSpd <-> Channel 2/fb_AT1K0_GAS_PTM_140.i_xAtSpd
//     PlcTask Inputs/GVL_Devices.fb_AT1K0_GAS_PTM_140.i_xDecel <-> Channel 1/fb_AT1K0_GAS_PTM_140.i_xDecel
//     PlcTask Inputs/GVL_Devices.fb_AT1K0_GAS_PTM_140.i_xNCFault <-> Channel 3/fb_AT1K0_GAS_PTM_140.i_xNCFault
//     PlcTask Inputs/GVL_Devices.fb_AT1K0_GAS_PTM_140.i_xRotate <-> Channel 4/fb_AT1K0_GAS_PTM_140.i_xRotate
//   plc_kfe_gatt Instance <-> =+-CX2020/EtherCAT1/=+-EK1100_06_00/=+-ES1004_06_19
//     PlcTask Inputs/GVL_Devices.fb_AT1K0_GAS_PTM_140.i_xAccel <-> Channel 1/fb_AT1K0_GAS_PTM_140.i_xAccel
//   plc_kfe_gatt Instance <-> =+-CX2020/EtherCAT1/=+-EK1100_06_00/=+-ES1088_06_20
//     PlcTask Inputs/GVL_Devices.fb_AT1K0_GAS_PMF_90.i_xAlarmOK <-> Channel 4/fb_AT1K0_GAS_PMF_90.i_xAlarmOK
//     PlcTask Inputs/GVL_Devices.fb_AT1K0_GAS_PMF_90.i_xBPStatus <-> Channel 2/fb_AT1K0_GAS_PMF_90.i_xBPStatus
//     PlcTask Inputs/GVL_Devices.fb_AT1K0_GAS_PMF_90.i_xMPStatus <-> Channel 1/fb_AT1K0_GAS_PMF_90.i_xMPStatus
//     PlcTask Inputs/GVL_Devices.fb_AT1K0_GAS_PMF_90.i_xRemote <-> Channel 5/fb_AT1K0_GAS_PMF_90.i_xRemote
//     PlcTask Inputs/GVL_Devices.fb_AT1K0_GAS_PMF_90.i_xWarning <-> Channel 3/fb_AT1K0_GAS_PMF_90.i_xWarning
//   plc_kfe_gatt Instance <-> =+-CX2020/EtherCAT1/=+-EK1100_06_00/=+-ES1088_06_23
//     PlcTask Inputs/GVL_Devices.fb_AT1K0_GAS_PMF_100.i_xAlarmOK <-> Channel 4/fb_AT1K0_GAS_PMF_100.i_xAlarmOK
//     PlcTask Inputs/GVL_Devices.fb_AT1K0_GAS_PMF_100.i_xBPStatus <-> Channel 2/fb_AT1K0_GAS_PMF_100.i_xBPStatus
//     PlcTask Inputs/GVL_Devices.fb_AT1K0_GAS_PMF_100.i_xMPStatus <-> Channel 1/fb_AT1K0_GAS_PMF_100.i_xMPStatus
//     PlcTask Inputs/GVL_Devices.fb_AT1K0_GAS_PMF_100.i_xRemote <-> Channel 5/fb_AT1K0_GAS_PMF_100.i_xRemote
//     PlcTask Inputs/GVL_Devices.fb_AT1K0_GAS_PMF_100.i_xWarning <-> Channel 3/fb_AT1K0_GAS_PMF_100.i_xWarning
//   plc_kfe_gatt Instance <-> =+-CX2020/EtherCAT1/=+-EK1100_06_00/=+-ES3064_06_04
//     PlcTask Inputs/GVL_Devices.fb_AT1K0_GAS_PTM_110.i_iRawSpeed <-> AI Standard Channel 1/fb_AT1K0_GAS_PTM_110.i_iRawSpeed
//   plc_kfe_gatt Instance <-> =+-CX2020/EtherCAT1/=+-EK1100_06_00/=+-ES3064_06_06
//     PlcTask Inputs/GVL_Devices.fb_AT1K0_GAS_PTM_120.i_iCurrentMon <-> AI Standard Channel 2/fb_AT1K0_GAS_PTM_120.i_iCurrentMon
//     PlcTask Inputs/GVL_Devices.fb_AT1K0_GAS_PTM_120.i_iRawSpeed <-> AI Standard Channel 1/fb_AT1K0_GAS_PTM_120.i_iRawSpeed
//     PlcTask Inputs/GVL_Devices.fb_AT1K0_GAS_PTM_120.i_iTempMon <-> AI Standard Channel 3/fb_AT1K0_GAS_PTM_120.i_iTempMon
//   plc_kfe_gatt Instance <-> =+-CX2020/EtherCAT1/=+-EK1100_06_00/=+-ES3064_06_14
//     PlcTask Inputs/GVL_Devices.fb_AT1K0_GAS_PTM_130.i_iCurrentMon <-> AI Standard Channel 2/fb_AT1K0_GAS_PTM_130.i_iCurrentMon
//     PlcTask Inputs/GVL_Devices.fb_AT1K0_GAS_PTM_130.i_iRawSpeed <-> AI Standard Channel 1/fb_AT1K0_GAS_PTM_130.i_iRawSpeed
//     PlcTask Inputs/GVL_Devices.fb_AT1K0_GAS_PTM_130.i_iTempMon <-> AI Standard Channel 3/fb_AT1K0_GAS_PTM_130.i_iTempMon
//   plc_kfe_gatt Instance <-> =+-CX2020/EtherCAT1/=+-EK1100_06_00/=+-ES3064_06_16
//     PlcTask Inputs/GVL_Devices.fb_AT1K0_GAS_PTM_140.i_iCurrentMon <-> AI Standard Channel 2/fb_AT1K0_GAS_PTM_140.i_iCurrentMon
//     PlcTask Inputs/GVL_Devices.fb_AT1K0_GAS_PTM_140.i_iRawSpeed <-> AI Standard Channel 1/fb_AT1K0_GAS_PTM_140.i_iRawSpeed
//     PlcTask Inputs/GVL_Devices.fb_AT1K0_GAS_PTM_140.i_iTempMon <-> AI Standard Channel 3/fb_AT1K0_GAS_PTM_140.i_iTempMon
//   plc_kfe_gatt Instance <-> =+-CX2020/EtherCAT1/=+-EK1100_06_00/=+-ES4004_06_05
//     PlcTask Outputs/GVL_Devices.fb_AT1K0_GAS_PTM_110.q_iSpeedSet <-> AO Outputs Channel 1/fb_AT1K0_GAS_PTM_110.q_iSpeedSet
//     PlcTask Outputs/GVL_Devices.fb_AT1K0_GAS_PTM_120.q_iSpeedSet <-> AO Outputs Channel 3/fb_AT1K0_GAS_PTM_120.q_iSpeedSet
//   plc_kfe_gatt Instance <-> =+-CX2020/EtherCAT1/=+-EK1100_06_00/=+-ES4004_06_15
//     PlcTask Outputs/GVL_Devices.fb_AT1K0_GAS_PTM_130.q_iSpeedSet <-> AO Outputs Channel 1/fb_AT1K0_GAS_PTM_130.q_iSpeedSet
//     PlcTask Outputs/GVL_Devices.fb_AT1K0_GAS_PTM_140.q_iSpeedSet <-> AO Outputs Channel 3/fb_AT1K0_GAS_PTM_140.q_iSpeedSet
//   plc_kfe_gatt Instance <-> =+-CX2020/EtherCAT1/=+-EK1200_00_00/=+-ES2202_00_07
//     PlcTask Outputs/GVL_ILK.g_FastFaultOutput1.q_xFastFaultOut <-> Channel 1/Output
//     PlcTask Outputs/GVL_ILK.g_FastFaultOutput2.q_xFastFaultOut <-> Channel 2/Output
//   plc_kfe_gatt Instance <-> NC-Task 1 SAF/Axes/MA_1_X
//     PlcTask Inputs/Main.M1.Axis.NcToPlc <-> Outputs/ToPlc
//     PlcTask Outputs/Main.M1.Axis.PlcToNc <-> Inputs/FromPlc
//   plc_kfe_gatt Instance <-> NC-Task 1 SAF/Axes/MA_1_Y
//     PlcTask Inputs/Main.M2.Axis.NcToPlc <-> Outputs/ToPlc
//     PlcTask Outputs/Main.M2.Axis.PlcToNc <-> Inputs/FromPlc
//   plc_kfe_gatt Instance <-> NC-Task 1 SAF/Axes/MA_2_X
//     PlcTask Inputs/Main.M3.Axis.NcToPlc <-> Outputs/ToPlc
//     PlcTask Outputs/Main.M3.Axis.PlcToNc <-> Inputs/FromPlc
//   plc_kfe_gatt Instance <-> NC-Task 1 SAF/Axes/MA_2_Y
//     PlcTask Inputs/Main.M4.Axis.NcToPlc <-> Outputs/ToPlc
//     PlcTask Outputs/Main.M4.Axis.PlcToNc <-> Inputs/FromPlc
//   plc_kfe_gatt Instance <-> NC-Task 1 SAF/Axes/MA_3_X
//     PlcTask Inputs/Main.M5.Axis.NcToPlc <-> Outputs/ToPlc
//     PlcTask Outputs/Main.M5.Axis.PlcToNc <-> Inputs/FromPlc
//   plc_kfe_gatt Instance <-> NC-Task 1 SAF/Axes/MA_3_Y
//     PlcTask Inputs/Main.M6.Axis.NcToPlc <-> Outputs/ToPlc
//     PlcTask Outputs/Main.M6.Axis.PlcToNc <-> Inputs/FromPlc
//   plc_kfe_gatt Instance <-> NC-Task 1 SAF/Axes/MA_4_X
//     PlcTask Inputs/Main.M7.Axis.NcToPlc <-> Outputs/ToPlc
//     PlcTask Outputs/Main.M7.Axis.PlcToNc <-> Inputs/FromPlc
//   plc_kfe_gatt Instance <-> NC-Task 1 SAF/Axes/MA_4_Y
//     PlcTask Inputs/Main.M8.Axis.NcToPlc <-> Outputs/ToPlc
//     PlcTask Outputs/Main.M8.Axis.PlcToNc <-> Inputs/FromPlc
//   plc_kfe_gatt Instance <-> NC-Task 1 SAF/Axes/VGP_80
//     PlcTask Inputs/GVL_Devices.VGP_80.Axis.NcToPlc <-> Outputs/ToPlc
//     PlcTask Outputs/GVL_Devices.VGP_80.Axis.PlcToNc <-> Inputs/FromPlc

// ---- GVLs/GVL_Devices.TcGVL
VAR_GLOBAL
(*AT1K0*)
/// Injector
//Valves
	{attribute 'pytmc' :=' pv: AT1K0:GAS:VCN:70 '}
	VCN_70 : FB_VCN;
	
	{attribute 'pytmc' :=' pv: AT1K0:GAS:VVC:71 '}
	VVC_71 : FB_VVC;

	{attribute 'pytmc' :=' pv: AT1K0:GAS:VVC:72 '}
	VVC_72 : FB_VVC;
	
		
	{attribute 'pytmc' :=' pv: AT1K0:GAS:VGP:80 '}
	VGP_80 : FB_VGP;

//Gauges	
	{attribute 'pytmc' :=' pv: AT1K0:GAS:GCM:70 '}
	GCM_70: FB_GCM;
	{attribute 'pytmc' :=' pv: AT1K0:GAS:GCM:80 '}
	GCM_80: FB_GCM;
	{attribute 'pytmc' :=' pv: AT1K0:GAS:GCM:81 '}
	GCM_81: FB_GCM;
	(*Pseudo gauge device Structure to combine the readings of two GCM gauges*)
	{attribute 'pytmc' :=' pv: AT1K0:GAS:GCM:82  '}
	GCM_82 : ST_VG;
	
	
/////////////////////////////
	
		
	//////////////////////////////////
// MKS275 Gauges

{attribute 'pytmc' := ' pv: AT1K0:GAS:GPI:111 '}
fb_AT1K0_GAS_GPI_111 : FB_MKS275;
{attribute 'pytmc' := ' pv: AT1K0:GAS:GPI:121 '}
fb_AT1K0_GAS_GPI_121 : FB_MKS275;
{attribute 'pytmc' := ' pv: AT1K0:GAS:GPI:141 '}
fb_AT1K0_GAS_GPI_141 : FB_MKS275;

// FB_MKS317

{attribute 'pytmc' := ' pv: AT1K0:GAS:GPI:10 '}
fb_AT1K0_GAS_GPI_10 : FB_MKS317;
{attribute 'pytmc' := ' pv: AT1K0:GAS:GPI:20 '}
fb_AT1K0_GAS_GPI_20 : FB_MKS317;
{attribute 'pytmc' := ' pv: AT1K0:GAS:GPI:11 '}
fb_AT1K0_GAS_GPI_11 : FB_MKS317;
{attribute 'pytmc' := ' pv: AT1K0:GAS:GPI:30 '}
fb_AT1K0_GAS_GPI_30 : FB_MKS317;
{attribute 'pytmc' := ' pv: AT1K0:GAS:GPI:40 '}
fb_AT1K0_GAS_GPI_40 : FB_MKS317;
{attribute 'pytmc' := ' pv: AT1K0:GAS:GPI:50 '}
fb_AT1K0_GAS_GPI_50 : FB_MKS317;
{attribute 'pytmc' := ' pv: AT1K0:GAS:GPI:60 '}
fb_AT1K0_GAS_GPI_60 : FB_MKS317;
{attribute 'pytmc' := ' pv: AT1K0:GAS:GPI:51 '}
fb_AT1K0_GAS_GPI_51 : FB_MKS317;
{attribute 'pytmc' := ' pv: AT1K0:GAS:GPI:80 '}
fb_AT1K0_GAS_GPI_80 : FB_MKS317;
{attribute 'pytmc' := ' pv: AT1K0:GAS:GPI:90 '}
fb_AT1K0_GAS_GPI_90 : FB_MKS317;
{attribute 'pytmc' := ' pv: AT1K0:GAS:GPI:100 '}
fb_AT1K0_GAS_GPI_100 : FB_MKS317;
{attribute 'pytmc' := ' pv: AT1K0:GAS:GPI:110 '}
fb_AT1K0_GAS_GPI_110 : FB_MKS317;
{attribute 'pytmc' := ' pv: AT1K0:GAS:GPI:120 '}
fb_AT1K0_GAS_GPI_120 : FB_MKS317;
{attribute 'pytmc' := ' pv: AT1K0:GAS:GPI:130 '}
fb_AT1K0_GAS_GPI_130 : FB_MKS317;
{attribute 'pytmc' := ' pv: AT1K0:GAS:GPI:140 '}
fb_AT1K0_GAS_GPI_140 : FB_MKS317;

// FB_MKS422

{attribute 'pytmc' := ' pv: AT1K0:GAS:GCC:10 '}
fb_AT1K0_GAS_GCC_10 : FB_MKS422;
{attribute 'pytmc' := ' pv: AT1K0:GAS:GCC:20 '}
fb_AT1K0_GAS_GCC_20 : FB_MKS422;
{attribute 'pytmc' := ' pv: AT1K0:GAS:GCC:30 '}
fb_AT1K0_GAS_GCC_30 : FB_MKS422;
{attribute 'pytmc' := ' pv: AT1K0:GAS:GCC:40 '}
fb_AT1K0_GAS_GCC_40 : FB_MKS422;
{attribute 'pytmc' := ' pv: AT1K0:GAS:GCC:50 '}
fb_AT1K0_GAS_GCC_50 : FB_MKS422;
{attribute 'pytmc' := ' pv: AT1K0:GAS:GCC:60 '}
fb_AT1K0_GAS_GCC_60 : FB_MKS422;
{attribute 'pytmc' := ' pv: AT1K0:GAS:GCC:80 '}
fb_AT1K0_GAS_GCC_80 : FB_MKS422;
{attribute 'pytmc' := ' pv: AT1K0:GAS:GCC:90 '}
fb_AT1K0_GAS_GCC_90 : FB_MKS422;
{attribute 'pytmc' := ' pv: AT1K0:GAS:GCC:100 '}
fb_AT1K0_GAS_GCC_100 : FB_MKS422;
{attribute 'pytmc' := ' pv: AT1K0:GAS:GCC:110 '}
fb_AT1K0_GAS_GCC_110 : FB_MKS422;
{attribute 'pytmc' := ' pv: AT1K0:GAS:GCC:120 '}
fb_AT1K0_GAS_GCC_120 : FB_MKS422;
{attribute 'pytmc' := ' pv: AT1K0:GAS:GCC:130 '}
fb_AT1K0_GAS_GCC_130 : FB_MKS422;
{attribute 'pytmc' := ' pv: AT1K0:GAS:GCC:140 '}
fb_AT1K0_GAS_GCC_140 : FB_MKS422;




// FB_VRC

{attribute 'pytmc' := ' pv: AT1K0:GAS:VRC:10 '}
fb_AT1K0_GAS_VRC_10 : FB_VRC_EBD;
{attribute 'pytmc' := ' pv: AT1K0:GAS:VRC:20 '}
fb_AT1K0_GAS_VRC_20 : FB_VRC_EBD;
{attribute 'pytmc' := ' pv: AT1K0:GAS:VRC:30 '}
fb_AT1K0_GAS_VRC_30 : FB_VRC_EBD;
{attribute 'pytmc' := ' pv: AT1K0:GAS:VRC:40 '}
fb_AT1K0_GAS_VRC_40 : FB_VRC_EBD;
{attribute 'pytmc' := ' pv: AT1K0:GAS:VRC:50 '}
fb_AT1K0_GAS_VRC_50 : FB_VRC;
{attribute 'pytmc' := ' pv: AT1K0:GAS:VRC:60 '}
fb_AT1K0_GAS_VRC_60 : FB_VRC;
{attribute 'pytmc' := ' pv: AT1K0:GAS:VRC:70 '}
fb_AT1K0_GAS_VRC_70 : FB_VRC;
{attribute 'pytmc' := ' pv: AT1K0:GAS:VRC:80 '}
fb_AT1K0_GAS_VRC_80 : FB_VRC;
{attribute 'pytmc' := ' pv: AT1K0:GAS:VRC:90 '}
fb_AT1K0_GAS_VRC_90 : FB_VRC;
{attribute 'pytmc' := ' pv: AT1K0:GAS:VRC:100 '}
fb_AT1K0_GAS_VRC_100 : FB_VRC;
{attribute 'pytmc' := ' pv: AT1K0:GAS:VRC:110 '}
fb_AT1K0_GAS_VRC_110 : FB_VRC;
{attribute 'pytmc' := ' pv: AT1K0:GAS:VRC:120 '}
fb_AT1K0_GAS_VRC_120 : FB_VRC;
{attribute 'pytmc' := ' pv: AT1K0:GAS:VRC:130 '}
fb_AT1K0_GAS_VRC_130 : FB_VRC;
{attribute 'pytmc' := ' pv: AT1K0:GAS:VRC:140 '}
fb_AT1K0_GAS_VRC_140 : FB_VRC;

// PUMPS
// Turbos
// FB_PTM_Ebara_010M
{attribute 'pytmc' := ' pv: AT1K0:GAS:PTM:10 '}
fb_AT1K0_GAS_PTM_10 : FB_PTM_Ebara_010M;
{attribute 'pytmc' := ' pv: AT1K0:GAS:PTM:20 '}
fb_AT1K0_GAS_PTM_20 : FB_PTM_Ebara_010M;
{attribute 'pytmc' := ' pv: AT1K0:GAS:PTM:30 '}
fb_AT1K0_GAS_PTM_30 : FB_PTM_Ebara_010M;
{attribute 'pytmc' := ' pv: AT1K0:GAS:PTM:40 '}
fb_AT1K0_GAS_PTM_40 : FB_PTM_Ebara_010M;
{attribute 'pytmc' := ' pv: AT1K0:GAS:PTM:80 '}
fb_AT1K0_GAS_PTM_80 : FB_PTM_TwisTorr;
{attribute 'pytmc' := ' pv: AT1K0:GAS:PTM:120 '}
fb_AT1K0_GAS_PTM_120 : FB_PTM_Ebara_010M;
{attribute 'pytmc' := ' pv: AT1K0:GAS:PTM:130 '}
fb_AT1K0_GAS_PTM_130 : FB_PTM_Ebara_010M;
{attribute 'pytmc' := ' pv: AT1K0:GAS:PTM:140 '}
fb_AT1K0_GAS_PTM_140 : FB_PTM_Ebara_010M;
// FB_PTM_Ebara_011M
{attribute 'pytmc' := ' pv: AT1K0:GAS:PTM:110 '}
fb_AT1K0_GAS_PTM_110 : FB_PTM_Ebara_011M;

// Roughing
// FB_EbaraDryPump
{attribute 'pytmc' := ' pv: AT1K0:GAS:PMF:10 '}
fb_AT1K0_GAS_PMF_10 : FB_ScrollPump;
{attribute 'pytmc' := ' pv: AT1K0:GAS:PMF:60 '}
fb_AT1K0_GAS_PMF_60 : FB_ScrollPump;
{attribute 'pytmc' := ' pv: AT1K0:GAS:PMF:90 '}
fb_AT1K0_GAS_PMF_90 : FB_EbaraDryPump;
{attribute 'pytmc' := ' pv: AT1K0:GAS:PMF:100 '}
fb_AT1K0_GAS_PMF_100 : FB_EbaraDryPump;
{attribute 'pytmc' := ' pv: AT1K0:GAS:PMF:110 '}
fb_AT1K0_GAS_PMF_110 : FB_EbaraEVA;
{attribute 'pytmc' := ' pv: AT1K0:GAS:PMF:120 '}
fb_AT1K0_GAS_PMF_120 : FB_EbaraEVA;
{attribute 'pytmc' := ' pv: AT1K0:GAS:PMF:140 '}
fb_AT1K0_GAS_PMF_140 : FB_EbaraEVA;

//Roughing DC Valves
{attribute 'pytmc' := ' pv: AT1K0:GAS:VCP:110 '}
{attribute 'TcLinkTo' := 	'.q_xOPN_DO	:=	TIIB[=+-EL2212_06_25]^DOX Control Channel 1^Control^Output'}
fb_AT1K0_GAS_VVC_110 : FB_VVC;
{attribute 'pytmc' := ' pv: AT1K0:GAS:VCP:120 '}
{attribute 'TcLinkTo' := 	'.q_xOPN_DO	:=	TIIB[=+-EL2212_06_25]^DOX Control Channel 2^Control^Output'}
fb_AT1K0_GAS_VVC_120 : FB_VVC;
{attribute 'pytmc' := ' pv: AT1K0:GAS:VCP:140 '}
{attribute 'TcLinkTo' := 	'.q_xOPN_DO	:=	TIIB[=+-EL2212_06_26]^DOX Control Channel 1^Control^Output'}
fb_AT1K0_GAS_VVC_140 : FB_VVC;

//PTM 80 VRC back stream valve
{attribute 'pytmc' := ' pv: AT1K0:GAS:VVC:80 '}
{attribute 'TcLinkTo' := 	'.q_xOPN_DO	:=	TIIB[=+-EL2212_06_26]^DOX Control Channel 2^Control^Output'}
fb_AT1K0_GAS_VVC_80 : FB_VVC;

END_VAR

// ---- GVLs/GVL_ILK.TcGVL
VAR_GLOBAL
	
//MPS
{attribute 'pytmc' := '
    pv: plc:lfe:gatt:FF1
    '}
    {attribute 'TcLinkTo' := '.q_xFastFaultOut:=TIIB[=+-ES2202_00_07]^Channel 1^Output'}
    g_FastFaultOutput1  :   FB_HardwareFFOutput;
	
	{attribute 'pytmc' := '
    pv: plc:lfe:gatt:FF2
    '}
    {attribute 'TcLinkTo' := '.q_xFastFaultOut:=TIIB[=+-ES2202_00_07]^Channel 2^Output'}
    g_FastFaultOutput2  :   FB_HardwareFFOutput;
	
	{attribute 'pytmc' := '
    pv: plc:kfe:FF_RESET
    '}
    xFastFaultReset :   BOOL;



	{attribute 'pytmc' := 'pv: AT1K0:GAS:VAC:OVRD_ON'}
	xSystemOverrideMode	:	BOOL; (* Global system override for the GATT*)


(* Interlock related bits, local to the PLC*)
	US_MAA_OK:  BOOL;
	US_Turbo_Valves_Open:  BOOL;
	DS_MAA_OK: BOOL;
	DS_Turbo_Valves_Open:  BOOL;
	US_Turbo_Running:  BOOL;
	DS_Turbo_Running:  BOOL;
	TwinscrewPumps_Valves_Closed: BOOL;
	US_Roughing_Valves_Open : BOOL;
	DS_Roughing_Valves_Open : BOOL;
	US_Aperture_Closed: BOOL;
	DS_Aperture_Closed: BOOL;
	
	xUSAperturesOpnOK : BOOL;
	xDSAperturesOpnOK : BOOL;
	
END_VAR

// ---- POUs/FB_VGP.TcPOU
(* This function implements the Basic functions for the Vat Motorized valve*)
FUNCTION_BLOCK FB_VGP
VAR_INPUT
	i_xExtIlkOK	:	BOOL; //External Interlock, SET to TRUE if not used
	i_xOpenIlkOK: BOOL; //Interlock Bit that allows the valve to open
	i_xCloseIlkOK: BOOL; //Interlock Bit that allows the valve to Close
	
	i_ReqPos	:	REAL; //Requested position
	
	arrTable	: ARRAY[1..14,1..2] OF FLOAT;
END_VAR
VAR_OUTPUT
	{attribute 'pytmc' := '
    pv:
	'}
	q_stVGP	:	ST_VGP; // valve structure
END_VAR
VAR_IN_OUT
	
END_VAR

VAR CONSTANT
	
	rClosePosition : REAL:=0; // Encoder Min. Fully Closed
	rMaxDiffPressure: REAL:= 22.5; //Torr
END_VAR

VAR
	rOpenPosition: REAL:=1645; // Encoder MAX. Fully Open
	rTargetPosition : REAL;
	rTargetVelocity: REAL:=30;
	rHomingVelocity: REAL:=10;
	rHomingDistance: REAL:=20;//every 150 is 10% , 1%  is 14.975
	rOldTargetPosition: REAL;
		
	// 
	/// axis reference data structure 
	Axis: AXIS_REF;
	//
	InfoData_State AT %I*: UINT ;
	
	// Axis MC functions

	fbPowerAxis: MC_Power;
	/// debug function block output data 
	PowerAxisOut: ST_McOutputs;
	fbMoveAxisABS: MC_MoveAbsolute;
	/// debug function block output data 
	MoveAbsoluteOut: ST_McOutputs;
	fbMoveAxisABS2: MC_MoveAbsolute;
	/// debug function block output data 
	MoveAbsoluteOut2: ST_McOutputs;
	
	fbReset: MC_Reset;
	/// debug function block output data 
	ResetOut: ST_McOutputs;
	MoveAxisREL: MC_MoveAbsolute;
	MoveRelativeOut: ST_McOutputs;
	
	
	nErrorID: UDINT;
	bError : Bool;
	sErrorMessage : STRING;
	rOverride: LREAL := 100;
	fbHalt: MC_Halt;
	
	
	// Homing Functions
	bGo:BOOL := FALSE; //to execute motion
	bHome:BOOL :=FALSE; // should be set to true
	bEnable:Bool; //to be removed
	fbMoveRel: MC_MoveRelative;
	fbSetPosition: MC_SetPosition;
	fbWriteParameter: MC_WriteBoolParameter;
	HomeState: E_HomeState;
	
	
	// interpolation
	bInit : BOOL := TRUE;
	eMode           : E_CTRL_MODE;
	iCounter:INT;
	//CONTROL
	stCTRL_LIN_INTERPOLATION_PARAMS		: ST_CTRL_LIN_INTERPOLATION_PARAMS;
	fbCTRL_LIN_INTERPOLATION					: FB_CTRL_LIN_INTERPOLATION;
	arrTable_ENC : ARRAY[1..14,1..2] OF FLOAT;
	//Readdback
	stCTRL_LIN_INTERPOLATION_PARAMS_ENC		: ST_CTRL_LIN_INTERPOLATION_PARAMS;
	fbCTRL_LIN_INTERPOLATION_ENC					: FB_CTRL_LIN_INTERPOLATION;

END_VAR

/// Interpolation  function initialization
ACT_INIT();

// Interlocking
q_stVGP.xIlkOK := i_xExtIlkOK;
(*Checking which Control mode is selected*)
IF q_stVGP.xIlkOK AND NOT (q_stVGP.pv_xError) THEN
	IF q_stVGP.eValveControl = OpenValve THEN
		q_stVGP.rReqPosition := q_stVGP.rUpperLimit;
	ELSIF q_stVGP.eValveControl = CloseValve THEN
		q_stVGP.rReqPosition := 0;
	ELSIF q_stVGP.eValveControl = ManualControl THEN
		q_stVGP.rReqPosition := LIMIT(0, q_stVGP.rReqPosition, q_stVGP.rUpperLimit);
	ELSIF q_stVGP.eValveControl = PressureControl THEN
		 q_stVGP.rReqPosition := LIMIT(0, i_ReqPos, q_stVGP.rUpperLimit);
	END_IF
ELSE
	q_stVGP.rReqPosition := 0;
	q_stVGP.eValveControl := CloseValve;//CloseValve;
	bGo:=FALSE;
END_IF


//Check the Drive State

IF (*(InfoData_State<>16#8) OR*) (q_stVGP.state = MOVESTATE_ERROR) THEN
	q_stVGP.pv_xError:=TRUE;
ELSE
	q_stVGP.pv_xError:=FALSE;
	// Call function to execute move
	// call motion function blocks???
END_IF


IF (q_stVGP.pv_xABORT_SW ) THEN
	q_stVGP.pv_xABORT_SW := FALSE;
	q_stVGP.state:= MOVESTATE_ABORT;
END_IF


ACT_LIN_INTERPOLATION();
ACT_AXIS();
//ACT_HOME();

ACTION ACT_AXIS:
//update the axis status
AXIS();
q_stVGP.rEnoder_Position := LREAL_TO_REAL(Axis.NcToPlc.ActPos); // encoder position


IF NOT (i_xExtIlkOK) THEN
	q_stVGP.state := MOVESTATE_NEWTARGETPOSITION;
END_IF
//Homing STATE is missing

// state machine for axis motion
	(* move axis using a state machine *)
	CASE q_stVGP.state OF

		MOVESTATE_INIT :	(* initialisation *)
			(* initialize all function blocks *)
			fbMoveAxisABS.Execute := FALSE;
			fbMoveAxisABS2.Execute := FALSE;
			fbReset.Execute := FALSE;
			fbHALT.Execute :=FALSE;//
			q_stVGP.state := MOVESTATE_ENABLE; // Check homing first

		MOVESTATE_ENABLE :
			fbPowerAxis.Enable :=  TRUE;
			fbPowerAxis.Enable_Positive := TRUE;
			fbPowerAxis.Enable_Negative := TRUE;
			IF fbPowerAxis.Status THEN
				q_stVGP.state := MOVESTATE_READY;
			ELSIF fbPowerAxis.Error THEN
				q_stVGP.state := MOVESTATE_ERROR;
			END_IF
		
		MOVESTATE_READY: // waiting for move command
			IF (HomeState = READY) AND (q_stVGP.pv_xHome_SW) THEN
					HomeState:= INIT;
					q_stVGP.pv_xHome_SW:=false;
					bHome := false;
					q_stVGP.state := MOVESTATE_HOME;
					ELSE 
					q_stVGP.state := MOVESTATE_READY;
				END_IF
			IF (q_stVGP.pv_xGo_SW) AND i_xExtIlkOK(* AND( rOldTargetPosition <> rTargetPosition) *) THEN
				q_stVGP.pv_xGo_SW := false;
				q_stVGP.state := MOVESTATE_NEWTARGETPOSITION;	
			END_IF
			IF NOT fbPowerAxis.Status THEN
				q_stVGP.state := MOVESTATE_ENABLE;
			ELSIF fbPowerAxis.Error THEN
				q_stVGP.state := MOVESTATE_ERROR;
			END_IF
			
		MOVESTATE_HOME:
				if (HomeState = DONE) THEN
					 q_stVGP.state := MOVESTATE_READY;
					 q_stVGP.pv_xHomed := TRUE;
				END_IF
				
				if (HomeState = ERROR) THEN
					 q_stVGP.state := MOVESTATE_ERROR;
					  q_stVGP.pv_xHomed := FALSE;
				END_IF
				
		MOVESTATE_NEWTARGETPOSITION:
			fbMoveAxisABS.Position := rTargetPosition;	
			fbMoveAxisABS.Velocity := rTargetVelocity;		
			//fbMoveAxisABS.BufferMode := MC_BlendingNext;
			fbMoveAxisABS.Execute := TRUE;
			IF fbMoveAxisABS.Active  THEN
				(* axis is executing job but is not yet finished *)
				fbMoveAxisABS.Execute := FALSE;
				(* leave this state and buffer a second command *)
				q_stVGP.state := MOVESTATE_MOVING; 
			ElSIF fbMoveAxisABS.Done THEN
				fbMoveAxisABS.Execute := FALSE;
				q_stVGP.state := MOVESTATE_READY;
			ELSIF fbMoveAxisABS.CommandAborted OR fbMoveAxisABS.Error THEN
				q_stVGP.state := MOVESTATE_ERROR;
			END_IF
			
				
		MOVESTATE_MOVING://
			IF fbMoveAxisABS.CommandAborted OR fbMoveAxisABS.Error THEN
				q_stVGP.state := MOVESTATE_ERROR;
			END_IF	
			IF NOT ( Axis.Status.Moving) OR (fbMoveAxisABS.Done) THEN //(fbMoveAxisABS.Done) AND (fbMoveAxisABS2.Done) THEN
				q_stVGP.state := MOVESTATE_READY;	
			END_IF
			
		
		MOVESTATE_HALT:
			fbHALT.Execute :=TRUE;
			IF Axis.Status.Error THEN
				q_stVGP.state := MOVESTATE_RESET;	(* axis error requires reset *)
			ELSE
				q_stVGP.state := MOVESTATE_INIT;		(* function block errors don't need a reset *)
			END_IF
		
		MOVESTATE_ERROR :
			
			IF Axis.Status.Error THEN
				q_stVGP.state := MOVESTATE_RESET;	(* axis error requires reset *)
			ELSE
				q_stVGP.state := MOVESTATE_INIT;		(* function block errors don't need a reset *)
			END_IF

		MOVESTATE_RESET :
			fbReset.Execute := TRUE;
			IF fbReset.Done THEN
				q_stVGP.state := MOVESTATE_INIT;
			ELSIF fbReset.Error THEN
				q_stVGP.state := MOVESTATE_ERROR; (* keep trying to reset*)
			END_IF
			
		MOVESTATE_ABORT:
			fbMoveAxisABS.Execute := FALSE;
			fbMoveAxisABS2.Execute := FALSE;
			fbReset.Execute := FALSE;
			(* save target position*)
			rOldTargetPosition := 	q_stVGP.i_iPosition;
			fbHALT.Execute :=FALSE;
			fbPowerAxis.Enable := FALSE;
			fbPowerAxis.Enable_Positive := FALSE;
			fbPowerAxis.Enable_Negative := FALSE;
			q_stVGP.state := MOVESTATE_ENABLE; // Check homing first

	END_CASE





	
/// Motion Function Blocks
(* AXIS POWER*)
fbPowerAxis(
	Axis:= Axis, 
	Enable:= , 
	Enable_Positive:= i_xOpenIlkOK, 
	Enable_Negative:= , 
	Override:= rOverride, 
	BufferMode:= , 
	Options:= , 
	Status=>  , 
	Busy=> PowerAxisOut.Busy , 
	Active=> PowerAxisOut.Active , 
	Error=> PowerAxisOut.Error, 
	ErrorID=> PowerAxisOut.ErrorID);
(* AXIS MOVE ABSOLUTE*)
fbMoveAxisABS(
	Axis:= Axis , 
	Execute:= , 
	Position:= , 
	Velocity:= , 
	Acceleration:= , 
	Deceleration:= , 
	Jerk:= , 
	BufferMode:= MC_BlendingNext , 
	Options:= , 
	Done=>MoveAbsoluteOut.Done, 
	Busy=> MoveAbsoluteOut.Busy, 
	Active=> MoveAbsoluteOut.Active, 
	CommandAborted=> MoveAbsoluteOut.CommandAborted , 
	Error=> MoveAbsoluteOut.Error, 
	ErrorID=> MoveAbsoluteOut.ErrorID);
	(* AXIS MOVE ABSOLUTE*)
fbMoveAxisABS2(
	Axis:= Axis , 
	Execute:= , 
	Position:= , 
	Velocity:= , 
	Acceleration:= , 
	Deceleration:= , 
	Jerk:= , 
	BufferMode:= MC_BlendingNext , 
	Options:= , 
	Done=>MoveAbsoluteOut2.Done, 
	Busy=> MoveAbsoluteOut2.Busy, 
	Active=> MoveAbsoluteOut2.Active, 
	CommandAborted=> MoveAbsoluteOut2.CommandAborted , 
	Error=> MoveAbsoluteOut2.Error, 
	ErrorID=> MoveAbsoluteOut2.ErrorID);
(*AXIS RESET*)
fbReset(
	Axis:= Axis, 
	Execute:= , 
	Done=>ResetOut.Done , 
	Busy=>ResetOut.Busy , 
	Error=> ResetOut.Error, 
	ErrorID=> ResetOut.ErrorID);
(*HALT*)
fbHalt(
	Axis:= Axis, 
	Execute:= , 
	Deceleration:= , 
	Jerk:= , 
	BufferMode:= MC_BlendingNext , 
	Options:= , 
	Done=> , 
	Busy=> , 
	Active=> , 
	CommandAborted=> , 
	Error=> , 
	ErrorID=> );
	

/// ERROR
IF Axis.Status.Error THEN
	q_stVGP.state := MOVESTATE_ERROR;	
END_IF;	
	
// Error Handling
if( fbPowerAxis.Error and fbPowerAxis.Active ) then 
	bError:= fbPowerAxis.Error;
	nErrorID:= fbPowerAxis.ErrorID;
END_IF
if( fbMoveAxisABS.Error and fbMoveAxisABS.Active ) then 
	bError:= fbMoveAxisABS.Error;
	nErrorID:= fbMoveAxisABS.ErrorID;
END_IF

(*Convert nErrorID to string*)
sErrorMessage:=WORD_TO_HEXSTR(in:=TO_WORD(nErrorID) , iPrecision:= 4, bLoCase:=0 );
END_ACTION

ACTION ACT_HOME:


CASE HomeState OF
	READY:
		fbSetPosition.Execute := FALSE;
		fbWriteParameter.Execute := FALSE;
		fbMoveRel.Execute := FALSE;
		
	INIT:
		// disable soft limits in order to be able to move the drive
		fbWriteParameter.ParameterNumber := MC_AxisParameter.EnableLimitNeg;//EnableLimitPos;// .EnableLimitNeg;
		fbWriteParameter.Value := FALSE;
		fbWriteParameter.Execute := TRUE;
		if (fbWriteParameter.Done) THEN
			fbWriteParameter.Execute := FALSE;
			HomeState:= MOVING; 
		END_IF

	MOVING:
		IF fbMoveRel.Done THEN
			fbMoveRel.Execute := TRUE;
		END_IF;
		IF fbMoveRel.Active  THEN
			(* axis is executing job but is not yet finished *)
			fbMoveRel.Execute := FALSE;
			HomeState := MOVING2;
		ElSIF fbMoveRel.Done THEN
			fbMoveRel.Execute := FALSE;
			HomeState := MOVING2;
		ELSIF fbMoveRel.CommandAborted OR fbMoveRel.Error THEN
			fbMoveRel.Execute := FALSE;
			HomeState := ERROR;
		END_IF
	
	MOVING2:
		IF fbMoveRel.Done THEN
			fbMoveRel.Execute := TRUE;
		END_IF;
		IF fbMoveRel.Active  THEN
			(* axis is executing job but is not yet finished *)
			fbMoveRel.Execute := FALSE;
			HomeState := MOVING;
		ElSIF fbMoveRel.Done THEN
			fbMoveRel.Execute := FALSE;
			HomeState := MOVING;
		ELSIF fbMoveRel.CommandAborted OR fbMoveRel.Error THEN
			fbMoveRel.Execute := FALSE;
			HomeState := CHECK;
		END_IF	

	
	CHECK:
		//Check position lag monitoring error
		if ( Axis.Status.ErrorID = 17245)THEN 
			// Set Current Position
			fbSetPosition.Position := 0; //rOpenPosition+rHomingDistance;
			fbSetPosition.Execute := TRUE;
			if ( fbSetPosition.Done ) THEN
				fbSetPosition.Execute := FALSE;
				HomeState:= WRITE;
			END_IF
		ELSE
			HomeState := ERROR;
		END_IF
	
	ERROR:
	
	
	WRITE:
	// Re Enable the Soft limits	
		fbWriteParameter.ParameterNumber := MC_AxisParameter.AxisEnMinSoftPosLimit;//AxisEnMaxSoftPosLimit;// .AxisEnMinSoftPosLimit;
		fbWriteParameter.Value := TRUE;
		fbWriteParameter.Execute := TRUE;
		if (fbWriteParameter.Done) THEN
			fbWriteParameter.Execute := FALSE;
			HomeState:= DONE; 
		END_IF
	
	DONE:
	// Homing DONE STATE 
	// should go back to closed zero position???

END_CASE

// Move Forward
fbMoveRel(
	Axis:= Axis , 
	Execute:= , 
	Distance:= rHomingDistance , 
	Velocity:= rHomingVelocity, 
	Acceleration:= , 
	Deceleration:= , 
	Jerk:= , 
	BufferMode:= MC_BlendingNext, 
	Options:= , 
	Done=> , 
	Busy=> , 
	Active=> , 
	CommandAborted=> , 
	Error=> , 
	ErrorID=> );
	
// Set Encoder Position
fbSetPosition(
	Axis:= Axis , 
	Execute:= , 
	Position:= 0 , 
	Mode:= , 
	Options:= , 
	Done=> , 
	Busy=> , 
	Error=> , 
	ErrorID=> );
	
// Write Parameters
fbWriteParameter(
	Axis:= Axis , 
	Execute:= , 
	ParameterNumber:= , 
	Value:= , 
	Done=> , 
	Busy=> , 
	Error=> , 
	ErrorID=> );
END_ACTION

ACTION ACT_INIT:
IF bInit THEN
	
(*
	(* init array with the interpolation points  *)
	(* 	fIn					 |		fOut		*)
	arrTable[1,1] := 0;			arrTable[1,2] := 0;
	arrTable[2,1] := 5;		    arrTable[2,2] := 135;
	arrTable[3,1] := 10;		arrTable[3,2] := 245;
	arrTable[4,1] :=  20;	    arrTable[4,2] := 405;
	arrTable[5,1] :=  30;	    arrTable[5,2] := 535;
	arrTable[6,1] := 40;		arrTable[6,2] := 689;
	arrTable[7,1] := 50;		arrTable[7,2] := 830;
	arrTable[8,1] := 60;	    arrTable[8,2] := 960;
	arrTable[9,1] := 70;	    arrTable[9,2] := 1095;
	arrTable[10,1] := 80;		arrTable[10,2] := 1225;
	arrTable[11,1] := 90;		arrTable[11,2] := 1415;
	arrTable[12,1] := 95;		arrTable[12,2] := 1495;
	arrTable[13,1] := 98;		arrTable[13,2] := 1559;
	arrTable[14,1] := 100;		arrTable[14,2] := 1645;
	*)
	
	(* init parameter struct *)
	stCTRL_LIN_INTERPOLATION_PARAMS.tCtrlCycleTime					:= T#10ms;
	stCTRL_LIN_INTERPOLATION_PARAMS.tTaskCycleTime					:= T#10ms;
	stCTRL_LIN_INTERPOLATION_PARAMS.nDataTable_NumberOfRows		:= INT_TO_UINT(14);

	(* set the addresses *)
	stCTRL_LIN_INTERPOLATION_PARAMS.pDataTable_ADR			:= ADR(arrTable);
	stCTRL_LIN_INTERPOLATION_PARAMS.nDataTable_SIZEOF		:= SIZEOF(arrTable);

	(* set the mode to ACTIVE --> normal operation *)
	eMode							:= eCTRL_MODE_ACTIVE;
	
	
	(* init array with the interpolation points  *)
	(* 	fIn					 |		fOut		*)
	 FOR iCounter:=1 TO 14 BY 1 DO
		arrTable_ENC[iCounter,1] := arrTable[iCounter,2];
		arrTable_ENC[iCounter,2] := arrTable[iCounter,1];		
	 END_FOR;
	(*
	arrTable_ENC[1,1] := 0;			arrTable_ENC[1,2] := 0;
	arrTable_ENC[2,1] := 135;		    arrTable_ENC[2,2] := 5;
	arrTable_ENC[3,1] := 245;		arrTable_ENC[3,2] := 10;
	arrTable_ENC[4,1] :=  405;	    arrTable_ENC[4,2] := 20;
	arrTable_ENC[5,1] :=  535;	    arrTable_ENC[5,2] := 30;
	arrTable_ENC[6,1] := 689;		arrTable_ENC[6,2] := 40;
	arrTable_ENC[7,1] := 830;		arrTable_ENC[7,2] := 50;
	arrTable_ENC[8,1] := 960;	    arrTable_ENC[8,2] := 60;
	arrTable_ENC[9,1] := 1095;	    arrTable_ENC[9,2] := 70;
	arrTable_ENC[10,1] := 1225;		arrTable_ENC[10,2] := 80;
	arrTable_ENC[11,1] := 1415;		arrTable_ENC[11,2] := 90;
	arrTable_ENC[12,1] := 1495;		arrTable_ENC[12,2] := 95;
	arrTable_ENC[13,1] := 1559;		arrTable_ENC[13,2] := 98;
	arrTable_ENC[14,1] := 1645;		arrTable_ENC[14,2] := 100;*)
	
	
	(* init parameter struct *)
	stCTRL_LIN_INTERPOLATION_PARAMS_ENC.tCtrlCycleTime					:= T#10ms;
	stCTRL_LIN_INTERPOLATION_PARAMS_ENC.tTaskCycleTime					:= T#10ms;
	stCTRL_LIN_INTERPOLATION_PARAMS_ENC.nDataTable_NumberOfRows		:= INT_TO_UINT(14);

	(* set the addresses *)
	stCTRL_LIN_INTERPOLATION_PARAMS_ENC.pDataTable_ADR			:= ADR(arrTable_ENC);
	stCTRL_LIN_INTERPOLATION_PARAMS_ENC.nDataTable_SIZEOF		:= SIZEOF(arrTable_ENC);
	
	(* reset the init flag *)
	bInit							:= FALSE;
	
END_IF;
END_ACTION

ACTION ACT_LIN_INTERPOLATION:

fbCTRL_LIN_INTERPOLATION(
	fIn:= q_stVGP.rReqPosition , 
	fManValue:= 0, 
	bExtrapolate:= , 
	eMode:= eMode, 
	fOut=> , 
	bInIsGreaterThanMaxElement=> , 
	bInIsLessThanMinElement=> , 
	eState=> , 
	eErrorId=> , 
	bError=> , 
	stParams:= stCTRL_LIN_INTERPOLATION_PARAMS );
	
// Target position Calculation
rTargetPosition := LREAL_TO_REAL(fbCTRL_LIN_INTERPOLATION.fOut);
//rTargetPosition := LIMIT(rClosePosition, rTargetPosition, rOpenPosition);	
	
fbCTRL_LIN_INTERPOLATION_ENC(
	fIn:= Axis.NcToPlc.ActPos , 
	fManValue:= 0, 
	bExtrapolate:= , 
	eMode:= eMode, 
	fOut=>  , 
	bInIsGreaterThanMaxElement=> , 
	bInIsLessThanMinElement=> , 
	eState=> , 
	eErrorId=> , 
	bError=> , 
	stParams:= stCTRL_LIN_INTERPOLATION_PARAMS_ENC );
q_stVGP.i_iPosition := LREAL_TO_REAL(fbCTRL_LIN_INTERPOLATION_ENC.fOut);
END_ACTION

METHOD ConfigEncoder : BOOL
VAR_INPUT
	EncoderMax: REAl; // Maximum encoder reading from fully closed to fully open
	invert: Bool; // Invert Encoder Counting Direction
END_VAR
VAR
	fbWriteParameter1: MC_WriteBoolParameter;
END_VAR
rOpenPosition := EncoderMax;

// fEncScaleFactor  -  AxisEncoderScalingFactor
 
// bEncIsInverse  -              
if (invert) THEN
	fbWriteParameter1.ParameterNumber :=  MC_AxisParameter.AxisEncoderDirectionInverse;
	fbWriteParameter1.Value := True;
END_IF

// Write Parameters
fbWriteParameter1(
	Axis:= Axis , 
	Execute:= , 
	ParameterNumber:= , 
	Value:= , 
	Done=> , 
	Busy=> , 
	Error=> , 
	ErrorID=> );
END_METHOD

METHOD M_INIT : BOOL
VAR_INPUT
	arrTable	: ARRAY[1..14,1..2] OF FLOAT;
	arrTable_ENC : ARRAY[1..14,1..2] OF FLOAT;
END_VAR
(* init array with the interpolation points  *)
	(* 	fIn					 |		fOut		*)
	arrTable[1,1] := 0;			arrTable[1,2] := 0;
	arrTable[2,1] := 5;		    arrTable[2,2] := 135;
	arrTable[3,1] := 10;		arrTable[3,2] := 245;
	arrTable[4,1] :=  20;	    arrTable[4,2] := 405;
	arrTable[5,1] :=  30;	    arrTable[5,2] := 535;
	arrTable[6,1] := 40;		arrTable[6,2] := 689;
	arrTable[7,1] := 50;		arrTable[7,2] := 830;
	arrTable[8,1] := 60;	    arrTable[8,2] := 960;
	arrTable[9,1] := 70;	    arrTable[9,2] := 1095;
	arrTable[10,1] := 80;		arrTable[10,2] := 1225;
	arrTable[11,1] := 90;		arrTable[11,2] := 1415;
	arrTable[12,1] := 95;		arrTable[12,2] := 1495;
	arrTable[13,1] := 98;		arrTable[13,2] := 1559;
	arrTable[14,1] := 100;		arrTable[14,2] := 1645;
	
	
	(* init parameter struct *)
	stCTRL_LIN_INTERPOLATION_PARAMS.tCtrlCycleTime					:= T#10ms;
	stCTRL_LIN_INTERPOLATION_PARAMS.tTaskCycleTime					:= T#10ms;
	stCTRL_LIN_INTERPOLATION_PARAMS.nDataTable_NumberOfRows		:= INT_TO_UINT(14);

	(* set the addresses *)
	stCTRL_LIN_INTERPOLATION_PARAMS.pDataTable_ADR			:= ADR(arrTable);
	stCTRL_LIN_INTERPOLATION_PARAMS.nDataTable_SIZEOF		:= SIZEOF(arrTable);

	(* set the mode to ACTIVE --> normal operation *)
	eMode							:= eCTRL_MODE_ACTIVE;
	
	
	(* init array with the interpolation points  *)
	(* 	fIn					 |		fOut		*)
	arrTable_ENC[1,1] := 0;			arrTable_ENC[1,2] := 0;
	arrTable_ENC[2,1] := 135;		    arrTable_ENC[2,2] := 5;
	arrTable_ENC[3,1] := 245;		arrTable_ENC[3,2] := 10;
	arrTable_ENC[4,1] :=  405;	    arrTable_ENC[4,2] := 20;
	arrTable_ENC[5,1] :=  535;	    arrTable_ENC[5,2] := 30;
	arrTable_ENC[6,1] := 689;		arrTable_ENC[6,2] := 40;
	arrTable_ENC[7,1] := 830;		arrTable_ENC[7,2] := 50;
	arrTable_ENC[8,1] := 960;	    arrTable_ENC[8,2] := 60;
	arrTable_ENC[9,1] := 1095;	    arrTable_ENC[9,2] := 70;
	arrTable_ENC[10,1] := 1225;		arrTable_ENC[10,2] := 80;
	arrTable_ENC[11,1] := 1415;		arrTable_ENC[11,2] := 90;
	arrTable_ENC[12,1] := 1495;		arrTable_ENC[12,2] := 95;
	arrTable_ENC[13,1] := 1559;		arrTable_ENC[13,2] := 98;
	arrTable_ENC[14,1] := 1645;		arrTable_ENC[14,2] := 100;
	
	
	(* init parameter struct *)
	stCTRL_LIN_INTERPOLATION_PARAMS_ENC.tCtrlCycleTime					:= T#10ms;
	stCTRL_LIN_INTERPOLATION_PARAMS_ENC.tTaskCycleTime					:= T#10ms;
	stCTRL_LIN_INTERPOLATION_PARAMS_ENC.nDataTable_NumberOfRows		:= INT_TO_UINT(14);

	(* set the addresses *)
	stCTRL_LIN_INTERPOLATION_PARAMS_ENC.pDataTable_ADR			:= ADR(arrTable_ENC);
	stCTRL_LIN_INTERPOLATION_PARAMS_ENC.nDataTable_SIZEOF		:= SIZEOF(arrTable_ENC);
END_METHOD

METHOD M_ValveControl : BOOL
VAR_INPUT
	state:E_VCN; // Close, Open, Pressure, Manual
END_VAR
q_stVGP.eValveControl := state;
END_METHOD

METHOD PUBLIC SetEncoderMax : BOOL
VAR_INPUT
	EncoderMax: REAl;
END_VAR
rOpenPosition := EncoderMax;
END_METHOD

END_FUNCTION_BLOCK

// ---- POUs/DIAGNOSTICS.TcPOU
PROGRAM DIAGNOSTICS
VAR
	//Change the PLC String Name to the actual PLC NAME
	sPLCName :STRING := 'PLC-KFE_GATT';
	//Link the sAMSNetID to the Etherat Master netID
	i_sAMSNetID AT %I*: AMSNETID;
	// DO NOT CHANGE
	sAMSNetID : STRING; //used for EPICS PV
	sLibVersion_LCLS_General : STRING;(* := stLibVersion_LCLS_General.sVersion*) ;
	fbEcatDiag:FB_EcatDiag;
	bAllSlaveStateGood : BOOL;
	bMasterStateGood :BOOL;
	iMasterState: WORD;
	sMasterState:STRING;
	nSlaveNumber : UINT;
	aiSlaveStates: ARRAY[1..256] OF BYTE;
	aEcSlaveInfo :  ARRAY[1..256] OF ST_EcDevice;
END_VAR

// Instaniating a call to the fbEcatDiag
fbEcatDiag(
	I_AMSNetId:=i_sAMSNetID , 
	i_xFirstPass:= _TaskInfo[1].FirstCycle, 
	q_xAllSlaveStatesGood=> bAllSlaveStateGood , 
	q_anTermStates=> aiSlaveStates, 
	q_xMasterStateGood=>bMasterStateGood , 
	q_nMasterState=> iMasterState, 
	q_sMasterState=> sMasterState , 
	q_astEcConfSlaveInfo=> aEcSlaveInfo , 
	q_nSlaves=> nSlaveNumber);

END_PROGRAM

// ---- POUs/FB_MAA.TcPOU
FUNCTION_BLOCK FB_MAA
VAR_IN_OUT
	stYStage: DUT_MotionStage;
	stXStage: DUT_MotionStage;
END_VAR
VAR_INPUT
	fAprt1: LREAL;
	fAprt2: LREAL;
	fAprt3: LREAL;
	fAprt4: LREAL;
END_VAR
VAR

	fbYStage: FB_MotionStage;
	fbXStage: FB_MotionStage;
	
	 {attribute 'pytmc' := '
        pv: STATE
        io: io
    '}
    fbStates: FB_MAA_States;
	
	fReticle: LREAL;
END_VAR

fbYStage(stMotionStage:=stYStage);
fbXStage(stMotionStage:=stXStage);

// All stages have no STO
stYStage.bHardwareEnable := TRUE;
stXStage.bHardwareEnable := TRUE;
// No PMPS yet
stYStage.bPowerSelf := TRUE;
stXStage.bPowerSelf := TRUE;


fbStates(
    stMotionStage:=stYStage,
    fAprt1:=fAprt1,
    fAprt2:=fAprt2,
    fAprt3:=fAprt3,
    fAprt4:=fAprt4);

END_FUNCTION_BLOCK

// ---- POUs/FB_MAA_States.TcPOU
FUNCTION_BLOCK FB_MAA_States
VAR_IN_OUT
	   stMotionStage: DUT_MotionStage;
END_VAR
VAR_INPUT
	  bEnable: BOOL;
    {attribute 'pytmc' := '
        pv: SET
        io: io
    '}
    enumSet: E_MAA_states;
    bStatesLock: BOOL;
	fAprt1: LREAL;
	fAprt2: LREAL;
	fAprt3: LREAL;
	fAprt4: LREAL;
END_VAR
VAR_OUTPUT
    bError: BOOL;
    sErrorMessage: STRING;
    bBusy: BOOL;
    bDone: BOOL;
    {attribute 'pytmc' := '
        pv: GET
        io: i
    '}
    enumGet: E_MAA_States;
END_VAR
VAR
    bInit: BOOL;
    arrStates: ARRAY[1..15] OF DUT_PositionState;
    nIter: INT;

    {attribute 'pytmc' := '
        pv:
        io: io
    '}
    fbStateManager: FB_PositionStateManager;

    fbLockAprt1: FB_PositionStateLock;
    fbLockAprt2: FB_PositionStateLock;
    fbLockAprt3: FB_PositionStateLock;
    fbLockAprt4: FB_PositionStateLock;
END_VAR
VAR CONSTANT
	
	fSmallDelta: LREAL := 0.01;
	fBigDelta: LREAL := 10;
	fMaxVelocity: LREAL := 20;
	fHighAccel: LREAL := 200;
	fLowAccel: LREAL := 25;
	
	
    fInDelta: LREAL := 0.1;
    fOutDelta: LREAL := 0.1;
    fInVelocity: LREAL := 5;
    fOutVelocity: LREAL := 5;
    fAccel: LREAL := 200;
    fOutDecel: LREAL := 25;
END_VAR

IF NOT bInit THEN
    bInit := FALSE;
    FOR nIter := 1 TO 4 DO
        arrStates[nIter].fDelta := fInDelta;
        arrStates[nIter].fVelocity := fInVelocity;
        arrStates[nIter].fAccel := fAccel;
        arrStates[nIter].fDecel := fAccel;
        arrStates[nIter].bLocked := bStatesLock;
        arrStates[nIter].bValid := TRUE;
        // TODO implement PMPS instead of doing this
        arrStates[nIter].bMoveOk := TRUE;
    END_FOR
    arrStates[1].sName := '5.5mm';
    arrStates[1].fPosition := fAprt1;
    arrStates[1].fDelta := fOutDelta;
    arrStates[1].fVelocity := fOutVelocity;
    arrStates[1].fDecel := fOutDecel;
    arrStates[2].sName := '8mm';
    arrStates[2].fPosition := fAprt2;
    arrStates[3].sName := '10mm';
    arrStates[3].fPosition := fAprt3;
    arrStates[4].sName := '12mm';
    arrStates[4].fPosition := fAprt4;
END_IF

fbLockAprt1(stPositionState := arrStates[1]);
fbLockAprt2(stPositionState := arrStates[2]);
fbLockAprt3(stPositionState := arrStates[3]);
fbLockAprt4(stPositionState := arrStates[4]);

fbStateManager(
    stMotionStage := stMotionStage,
    arrStates := arrStates,
    setState := enumSet,
    bEnable := bEnable,
    bError => bError,
    sErrorMessage => sErrorMessage,
    bBusy => bBusy,
    bDone => bDone,
    getState => enumGet);

END_FUNCTION_BLOCK

// ---- POUs/PRG_1_PlcTask.TcPOU
PROGRAM PRG_1_PlcTask
VAR

bDebug : Bool := TRUE;
fbLogHandler: FB_LogHandler;
	
END_VAR

(*Ethercat Diagnostics*)
DIAGNOSTICS();
// Vacuum and differential pumping
PRG_GATT();
// Injector
PRG_INJ();

if (NOT bDebug)Then
	// Functionblock for PTP motion between different appertures
	PRG_Motion();
	// Motorised valve
	PRG_VGP();
ELSE
	PRG_Motors_Test();
END_IF



//Logger
fbLogHandler();

END_PROGRAM

// ---- POUs/PRG_GATT.TcPOU
PROGRAM PRG_GATT
VAR
	
END_VAR



// GAUGES
// MKS275 Gauges
fb_AT1K0_GAS_GPI_111(PG=>);
fb_AT1K0_GAS_GPI_121(PG=>);
fb_AT1K0_GAS_GPI_141(PG=>);
// FB_MKS317
fb_AT1K0_GAS_GPI_10(PG=>);
fb_AT1K0_GAS_GPI_20(PG=>);
fb_AT1K0_GAS_GPI_11(PG=>);
fb_AT1K0_GAS_GPI_30(PG=>);
fb_AT1K0_GAS_GPI_40(PG=>);
fb_AT1K0_GAS_GPI_50(PG=>);
fb_AT1K0_GAS_GPI_51(PG=>);
fb_AT1K0_GAS_GPI_60(PG=>);
fb_AT1K0_GAS_GPI_80(PG=>);
fb_AT1K0_GAS_GPI_90(PG=>);
fb_AT1K0_GAS_GPI_100(PG=>);
fb_AT1K0_GAS_GPI_110(PG=>);
fb_AT1K0_GAS_GPI_120(PG=>);
fb_AT1K0_GAS_GPI_130(PG=>);
fb_AT1K0_GAS_GPI_140(PG=>);

// FB_MKS422

fb_AT1K0_GAS_GCC_10(PG := fb_AT1K0_GAS_GPI_10.PG);
fb_AT1K0_GAS_GCC_20(PG := fb_AT1K0_GAS_GPI_20.PG);
fb_AT1K0_GAS_GCC_30(PG := fb_AT1K0_GAS_GPI_30.PG);
fb_AT1K0_GAS_GCC_40(PG := fb_AT1K0_GAS_GPI_40.PG);
fb_AT1K0_GAS_GCC_50(PG := fb_AT1K0_GAS_GPI_50.PG);
fb_AT1K0_GAS_GCC_60(PG := fb_AT1K0_GAS_GPI_60.PG);
fb_AT1K0_GAS_GCC_80(PG := fb_AT1K0_GAS_GPI_80.PG);
fb_AT1K0_GAS_GCC_90(PG := fb_AT1K0_GAS_GPI_90.PG);
fb_AT1K0_GAS_GCC_100(PG := fb_AT1K0_GAS_GPI_100.PG);
fb_AT1K0_GAS_GCC_110(PG := fb_AT1K0_GAS_GPI_110.PG);
fb_AT1K0_GAS_GCC_120(PG := fb_AT1K0_GAS_GPI_120.PG);
fb_AT1K0_GAS_GCC_130(PG := fb_AT1K0_GAS_GPI_130.PG);
fb_AT1K0_GAS_GCC_140(PG := fb_AT1K0_GAS_GPI_140.PG);


